RoboDK station: kr30 cnc FIXED BY ALBERT 2.rdk

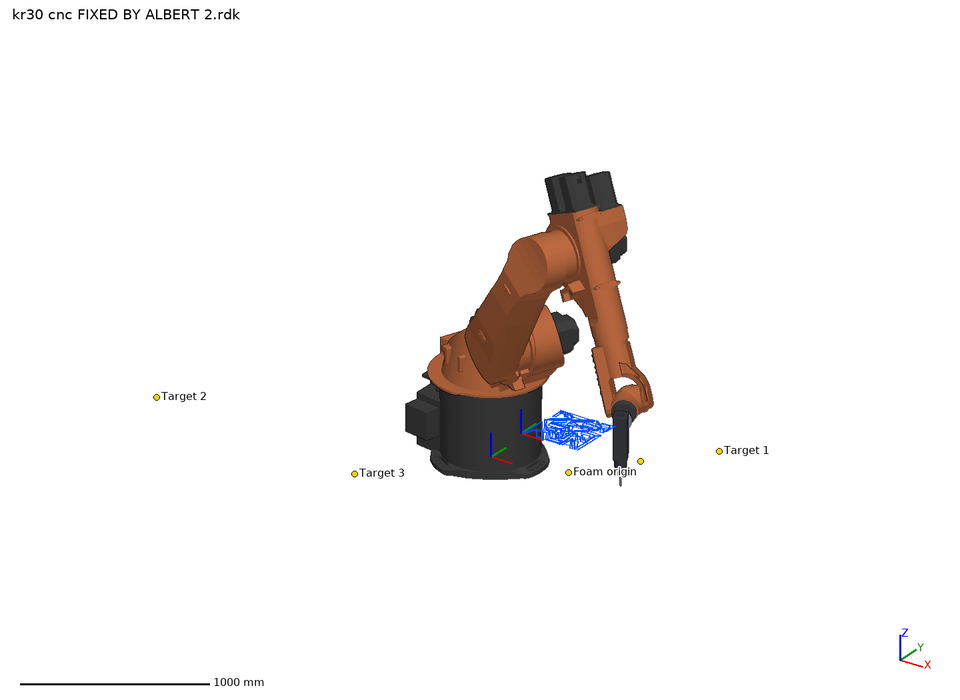
[picture v0: the station drawn from its stored meshes, robots at their saved joint values, targets as dots, program paths as lines]
Station kr30 cnc FIXED BY ALBERT 2. Poses are relative to the parent item; angles as X-Y-Z fixed-axis rotations.
  - frame KUKA KR 30 HA Base at (0, 0, 0) mm
    - robot KUKA KR 30 HA: 6 axes, payload 30 kg, reach 2033 mm, repeatability 0.05 mm, weight 665 kg
        modified DH rows (alpha deg, a mm, theta deg, d mm): 0, 0, 0, 815; -90, 350, 0, 0; 0, 850, -90, 0; -90, 145, 0, 820; 90, 0, 0, 0; -90, 0, 180, 170
        joint limits [-185, -135, -120, -350, -119, -350] to [185, 35, 158, 350, 119, 350]; home [0, -90, 90, 0, 0, 0]; saved at [21.032, -57.583, 122.737, -42.148, -71.052, 16.377]
      - tool 1/2" End Mill TCP, TCP at (337.71, -2.2, 160.57) mm, rotated rx 0 ry 90 rz 0 deg, size 415.8 x 102 x 153.6 mm
    - frame Reference Rhino at (909.29, -1020.53, 801.66) mm
      - object RhinoPart at (150, 150, -300) mm
      - target Target 1 (Cartesian target) at (994.45, 406.4, 10) mm, rotated rx 0 ry 90 rz -60.43 deg; joints [10.582, -19.112, 71.071, -56.398, -66.586, 30.882] of KUKA KR 30 HA
      - target Target 2 (Cartesian target) at (-1810.84, -765.32, 10.08) mm, rotated rx 49.23 ry 89.99 rz -110.09 deg; joints [109.49, -19.11, 71.06, -56.39, -66.58, 30.88] of KUKA KR 30 HA
      - target Target 3 (Cartesian target) at (-425.52, -920.6, 10.08) mm, rotated rx 49.23 ry 89.99 rz -69.31 deg; joints [68.71, -19.11, 71.06, -56.39, -66.58, 30.88] of KUKA KR 30 HA
      - target Foam origin (Cartesian target) at (180.49, 178.32, -252.76) mm, rotated rx -180 ry -0.01 rz -149.04 deg; joints [51.446, -59.335, 121.73, 83.267, -86.48, -27.398] of KUKA KR 30 HA
      - target Foam opposite corner (Cartesian target) at (416.08, 506.55, -249.15) mm, rotated rx -180 ry -0.01 rz -149.04 deg; joints [33.24, -61.647, 125.565, 66.534, -78.959, -23.784] of KUKA KR 30 HA
  - machining project RhinoPart Settings: C:/Users/Julian Ramirez.DESKTOP-JVDE542/Desktop/ELMER SHEET 1 TEST 3.nc | rotZ(0) | rotX(00)*rotY(360) | rotZ(0)
  - object box at (500, 500, 500) mm, size 250 x 250 x 250 mm, geometry from box.sld
  - program RhinoPart (818 instructions, listed below)
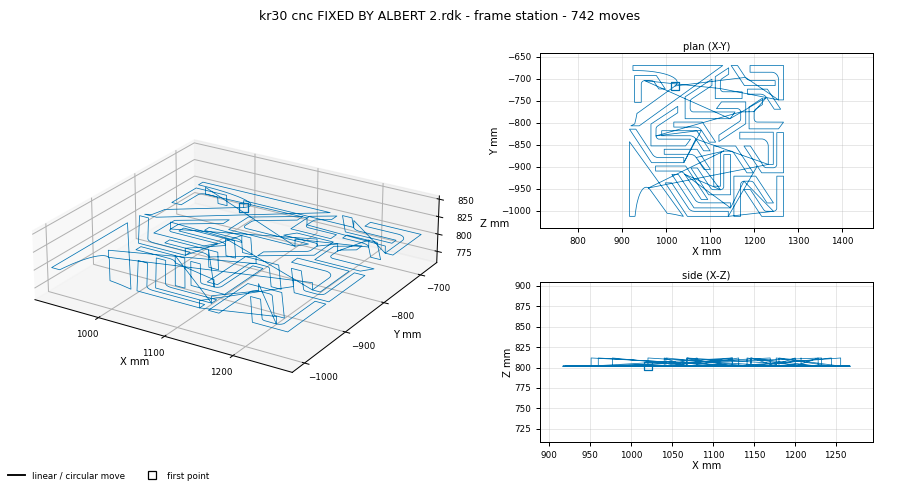
[picture p0: tool path of kr30 cnc FIXED BY ALBERT 2.rdk in frame station, 742 of 742 moves have a stored position in this frame; points joined in program order, loops and branches not executed]

--- program RhinoPart (robot KUKA KR 30 HA) ---
  Smooth(1)
  Set Ref.: Reference Rhino
  Set Tool: 1/2" End Mill TCP
  Show 1/2" End Mill TCP
  Set speed (2000.0 mm/s)
  MoveJ 1 to (111.39, 304.23, 0) mm, rotated rx -180 ry 0 rz 119.57 deg; joints [15.382, -66.233, 141.073, -46.061, -79.352, 10.854]
  MoveL 2 to (111.39, 304.23, 0) mm, rotated rx -180 ry 0 rz 119.57 deg; joints [15.382, -66.233, 141.073, -46.061, -79.352, 10.854]
  MoveL 3 to (111.39, 304.23, 0) mm, rotated rx -180 ry 0 rz 119.57 deg; joints [15.382, -66.233, 141.073, -46.061, -79.352, 10.854]
  Set speed (60.0 mm/s)
  MoveL 4 to (112.73, 305.44, 0) mm, rotated rx 180 ry 0 rz 119.57 deg; joints [15.298, -66.197, 141.001, -46.149, -79.343, 10.896]
  MoveL 5 to (113.84, 306.66, 0) mm, rotated rx -180 ry 0 rz 119.57 deg; joints [15.218, -66.168, 140.944, -46.233, -79.339, 10.931]
  MoveL 6 to (114.75, 307.89, 0) mm, rotated rx 180 ry 0 rz 119.57 deg; joints [15.14, -66.147, 140.903, -46.314, -79.34, 10.96]
  MoveL 7 to (115.44, 309.13, 0) mm, rotated rx 180 ry 0 rz 119.57 deg; joints [15.065, -66.134, 140.877, -46.39, -79.346, 10.983]
  MoveL 8 to (115.92, 310.36, 0) mm, rotated rx -180 ry 0 rz 119.57 deg; joints [14.993, -66.128, 140.867, -46.463, -79.356, 11.001]
  MoveL 9 to (116.19, 311.6, 0) mm, rotated rx -180 ry 0 rz 119.57 deg; joints [14.924, -66.13, 140.871, -46.532, -79.37, 11.012]
  MoveL 10 to (116.26, 312.84, 0) mm, rotated rx -180 ry 0 rz 119.57 deg; joints [14.858, -66.14, 140.89, -46.597, -79.389, 11.017]
  MoveL 11 to (116.12, 314.07, 0) mm, rotated rx -180 ry 0 rz 119.57 deg; joints [14.795, -66.157, 140.923, -46.657, -79.413, 11.017]
  MoveL 12 to (115.78, 315.3, 0) mm, rotated rx -180 ry 0 rz 119.57 deg; joints [14.735, -66.182, 140.972, -46.714, -79.441, 11.01]
  MoveL 13 to (115.23, 316.52, 0) mm, rotated rx -180 ry 0 rz 119.57 deg; joints [14.678, -66.213, 141.034, -46.767, -79.473, 10.998]
  MoveL 14 to (114.49, 317.73, 0) mm, rotated rx -180 ry 0 rz 119.57 deg; joints [14.624, -66.252, 141.111, -46.816, -79.509, 10.98]
  MoveL 15 to (113.55, 318.93, 0) mm, rotated rx 180 ry 0 rz 119.57 deg; joints [14.573, -66.299, 141.202, -46.86, -79.549, 10.956]
  MoveL 16 to (112.41, 320.12, 0) mm, rotated rx -180 ry 0 rz 119.57 deg; joints [14.526, -66.352, 141.307, -46.9, -79.593, 10.926]
  MoveL 17 to (111.07, 321.29, 0) mm, rotated rx 180 ry 0 rz 119.57 deg; joints [14.482, -66.412, 141.425, -46.937, -79.641, 10.891]
  MoveL 18 to (109.54, 322.44, 0) mm, rotated rx 180 ry 0 rz 119.57 deg; joints [14.442, -66.48, 141.557, -46.968, -79.693, 10.85]
  MoveL 19 to (106.83, 324.17, 0) mm, rotated rx 180 ry 0 rz 119.57 deg; joints [14.387, -66.595, 141.785, -47.008, -79.78, 10.776]
  MoveL 20 to (103.93, 325.72, 0) mm, rotated rx 180 ry 0 rz 119.57 deg; joints [14.343, -66.716, 142.023, -47.036, -79.867, 10.697]
  MoveL 21 to (100.95, 327.1, 0) mm, rotated rx 180 ry 0 rz 119.57 deg; joints [14.31, -66.839, 142.264, -47.054, -79.954, 10.615]
  MoveL 22 to (97.98, 328.3, 0) mm, rotated rx 180 ry 0 rz 119.57 deg; joints [14.286, -66.959, 142.5, -47.063, -80.038, 10.533]
  MoveL 23 to (91.45, 330.54, 0) mm, rotated rx -180 ry 0 rz 119.57 deg; joints [14.255, -67.22, 143.011, -47.062, -80.214, 10.352]
  MoveL 24 to (84.62, 332.44, 0) mm, rotated rx 180 ry 0 rz 119.57 deg; joints [14.246, -67.488, 143.537, -47.039, -80.391, 10.162]
  MoveL 25 to (77.71, 334.02, 0) mm, rotated rx 180 ry 0 rz 119.57 deg; joints [14.256, -67.755, 144.061, -46.998, -80.565, 9.97]
  MoveL 26 to (70.95, 335.3, 0) mm, rotated rx -180 ry 0 rz 119.57 deg; joints [14.28, -68.014, 144.569, -46.944, -80.73, 9.781]
  MoveL 27 to (64.72, 336.28, 0) mm, rotated rx -180 ry 0 rz 119.57 deg; joints [14.313, -68.251, 145.032, -46.883, -80.88, 9.608]
  MoveL 28 to (58.43, 337.12, 0) mm, rotated rx -180 ry 0 rz 119.57 deg; joints [14.357, -68.488, 145.496, -46.814, -81.028, 9.434]
  MoveL 29 to (52.12, 337.8, 0) mm, rotated rx -180 ry 0 rz 119.57 deg; joints [14.409, -68.723, 145.958, -46.735, -81.174, 9.259]
  MoveL 30 to (45.84, 338.35, 0) mm, rotated rx -180 ry 0 rz 119.57 deg; joints [14.47, -68.957, 146.414, -46.649, -81.317, 9.086]
  MoveL 31 to (39.9, 338.74, 0) mm, rotated rx 180 ry 0 rz 119.57 deg; joints [14.535, -69.176, 146.843, -46.561, -81.451, 8.922]
  MoveL 32 to (35.07, 338.99, 0) mm, rotated rx 180 ry 0 rz 119.57 deg; joints [14.593, -69.353, 147.189, -46.485, -81.558, 8.79]
  MoveL 33 to (30.23, 339.16, 0) mm, rotated rx 180 ry 0 rz 119.57 deg; joints [14.656, -69.53, 147.535, -46.404, -81.664, 8.657]
  MoveL 34 to (25.39, 339.26, 0) mm, rotated rx -180 ry 0 rz 119.57 deg; joints [14.724, -69.706, 147.878, -46.319, -81.77, 8.525]
  MoveL 35 to (20.56, 339.29, 0) mm, rotated rx 180 ry 0 rz 119.57 deg; joints [14.796, -69.881, 148.22, -46.23, -81.874, 8.393]
  MoveL 36 to (15.58, 339.29, 0) mm, rotated rx 180 ry 0 rz 119.57 deg; joints [14.873, -70.061, 148.57, -46.135, -81.981, 8.258]
  MoveL 37 to (15.58, 350.72, 0) mm, rotated rx -180 ry 0 rz 119.57 deg; joints [14.201, -70.168, 148.779, -46.796, -82.148, 8.276]
  MoveL 38 to (219.85, 350.72, 0) mm, rotated rx 180 ry 0 rz 119.57 deg; joints [11.685, -62.59, 133.888, -50.278, -77.793, 14.278]
  MoveL 39 to (29.95, 213.56, 0) mm, rotated rx 180 ry 0 rz 119.57 deg; joints [21.65, -68.069, 144.677, -39.552, -79.597, 8.481]
  MoveL 40 to (10.8, 213.56, 0) mm, rotated rx -180 ry 0 rz 119.57 deg; joints [22.063, -68.737, 145.985, -39.064, -80.033, 7.996]
  MoveL 41 to (19.53, 217.8, 0) mm, rotated rx -180 ry 0 rz 119.57 deg; joints [21.645, -68.492, 145.505, -39.51, -79.911, 8.22]
  MoveL 42 to (20.98, 223.68, 0) mm, rotated rx -180 ry 0 rz 119.57 deg; joints [21.296, -68.522, 145.564, -39.857, -79.983, 8.262]
  MoveL 43 to (22.33, 229.61, 0) mm, rotated rx 180 ry 0 rz 119.57 deg; joints [20.946, -68.555, 145.629, -40.206, -80.058, 8.303]
  MoveL 44 to (23.58, 235.57, 0) mm, rotated rx -180 ry 0 rz 119.57 deg; joints [20.597, -68.59, 145.698, -40.553, -80.134, 8.341]
  MoveL 45 to (24.71, 241.54, 0) mm, rotated rx 180 ry 0 rz 119.57 deg; joints [20.248, -68.629, 145.773, -40.899, -80.213, 8.376]
  MoveL 46 to (24.55, 241.81, 0) mm, rotated rx 180 ry 0 rz 119.57 deg; joints [20.236, -68.638, 145.791, -40.91, -80.221, 8.372]
  MoveL 47 to (25.65, 242.44, 0) mm, rotated rx -180 ry 0 rz 119.57 deg; joints [20.18, -68.608, 145.732, -40.97, -80.207, 8.402]
  MoveL 48 to (26.73, 243.1, 0) mm, rotated rx 180 ry 0 rz 119.57 deg; joints [20.122, -68.578, 145.674, -41.03, -80.194, 8.43]
  MoveL 49 to (27.79, 243.78, 0) mm, rotated rx 180 ry 0 rz 119.57 deg; joints [20.064, -68.55, 145.618, -41.092, -80.182, 8.458]
  MoveL 50 to (28.82, 244.5, 0) mm, rotated rx 180 ry 0 rz 119.57 deg; joints [20.004, -68.522, 145.565, -41.156, -80.172, 8.486]
  MoveL 51 to (109.85, 303.02, 0) mm, rotated rx 180 ry 0 rz 119.57 deg; joints [15.468, -66.278, 141.161, -45.969, -79.366, 10.807]
  MoveL 52 to (111.39, 304.23, 0) mm, rotated rx -180 ry 0 rz 119.57 deg; joints [15.382, -66.233, 141.073, -46.061, -79.352, 10.854]
  Set speed (2000.0 mm/s)
  MoveL 53 to (111.39, 304.23, 0) mm, rotated rx -180 ry 0 rz 119.57 deg; joints [15.382, -66.233, 141.073, -46.061, -79.352, 10.854]
  MoveL 54 to (111.39, 304.23, 10) mm, rotated rx -180 ry 0 rz 119.57 deg; joints [15.382, -67.039, 141.042, -46.178, -78.772, 11.469]
  Set speed (2000.0 mm/s)
  MoveL 55 to (271.36, 323.77, 0) mm, rotated rx 180 ry 0 rz 119.57 deg; joints [12.449, -60.385, 129.521, -49.903, -76.207, 15.81]
  MoveL 56 to (271.36, 323.77, 0) mm, rotated rx 180 ry 0 rz 119.57 deg; joints [12.449, -60.385, 129.521, -49.903, -76.207, 15.81]
  Set speed (60.0 mm/s)
  MoveL 57 to (253.54, 350.72, 0) mm, rotated rx -180 ry 0 rz 119.57 deg; joints [11.352, -61.296, 131.325, -50.826, -77.072, 15.353]
  MoveL 58 to (238.98, 350.72, 0) mm, rotated rx 180 ry 0 rz 119.57 deg; joints [11.494, -61.857, 132.437, -50.589, -77.384, 14.885]
  MoveL 59 to (269.2, 305, 0) mm, rotated rx 180 ry 0 rz 119.57 deg; joints [13.346, -60.302, 129.357, -49.029, -75.911, 15.659]
  MoveL 60 to (339.09, 305, 0) mm, rotated rx -180 ry 0 rz 119.57 deg; joints [12.617, -57.556, 123.906, -50.298, -74.371, 17.977]
  MoveL 61 to (339.09, 316.43, 0) mm, rotated rx 180 ry 0 rz 119.57 deg; joints [12.112, -57.656, 124.105, -50.776, -74.59, 18.032]
  MoveL 62 to (285.54, 316.43, 0) mm, rotated rx -180 ry 0 rz 119.57 deg; joints [12.643, -59.769, 128.3, -49.827, -75.764, 16.24]
  MoveL 63 to (284.51, 316.46, 0) mm, rotated rx 180 ry 0 rz 119.57 deg; joints [12.652, -59.81, 128.381, -49.81, -75.787, 16.206]
  MoveL 64 to (283.47, 316.55, 0) mm, rotated rx 180 ry 0 rz 119.57 deg; joints [12.659, -59.851, 128.462, -49.796, -75.811, 16.173]
  MoveL 65 to (282.45, 316.7, 0) mm, rotated rx 180 ry 0 rz 119.57 deg; joints [12.663, -59.892, 128.544, -49.784, -75.837, 16.14]
  MoveL 66 to (281.43, 316.91, 0) mm, rotated rx 180 ry 0 rz 119.57 deg; joints [12.664, -59.934, 128.626, -49.775, -75.863, 16.108]
  MoveL 67 to (280.43, 317.18, 0) mm, rotated rx -180 ry 0 rz 119.57 deg; joints [12.662, -59.975, 128.708, -49.769, -75.889, 16.076]
  MoveL 68 to (279.45, 317.5, 0) mm, rotated rx -180 ry 0 rz 119.57 deg; joints [12.657, -60.016, 128.79, -49.766, -75.917, 16.045]
  MoveL 69 to (278.48, 317.88, 0) mm, rotated rx 180 ry 0 rz 119.57 deg; joints [12.649, -60.057, 128.871, -49.766, -75.945, 16.016]
  MoveL 70 to (277.54, 318.32, 0) mm, rotated rx 180 ry 0 rz 119.57 deg; joints [12.638, -60.098, 128.951, -49.769, -75.974, 15.987]
  MoveL 71 to (276.62, 318.82, 0) mm, rotated rx -180 ry 0 rz 119.57 deg; joints [12.625, -60.138, 129.031, -49.775, -76.003, 15.959]
  MoveL 72 to (275.74, 319.38, 0) mm, rotated rx -180 ry 0 rz 119.57 deg; joints [12.608, -60.177, 129.108, -49.784, -76.032, 15.933]
  MoveL 73 to (274.9, 319.98, 0) mm, rotated rx 180 ry 0 rz 119.57 deg; joints [12.589, -60.215, 129.184, -49.797, -76.062, 15.908]
  MoveL 74 to (274.09, 320.64, 0) mm, rotated rx -180 ry 0 rz 119.57 deg; joints [12.566, -60.252, 129.257, -49.812, -76.091, 15.885]
  MoveL 75 to (273.34, 321.35, 0) mm, rotated rx 180 ry 0 rz 119.57 deg; joints [12.541, -60.287, 129.328, -49.83, -76.121, 15.863]
  MoveL 76 to (272.62, 322.11, 0) mm, rotated rx 180 ry 0 rz 119.57 deg; joints [12.513, -60.322, 129.395, -49.852, -76.15, 15.843]
  MoveL 77 to (271.96, 322.92, 0) mm, rotated rx 180 ry 0 rz 119.57 deg; joints [12.483, -60.354, 129.46, -49.876, -76.179, 15.826]
  MoveL 78 to (271.36, 323.77, 0) mm, rotated rx 180 ry 0 rz 119.57 deg; joints [12.449, -60.385, 129.521, -49.903, -76.207, 15.81]
  Set speed (2000.0 mm/s)
  MoveL 79 to (271.36, 323.77, 0) mm, rotated rx 180 ry 0 rz 119.57 deg; joints [12.449, -60.385, 129.521, -49.903, -76.207, 15.81]
  MoveL 80 to (271.36, 323.77, 10) mm, rotated rx -180 ry 0 rz 119.57 deg; joints [12.449, -61.047, 129.494, -50.035, -75.764, 16.354]
  Set speed (2000.0 mm/s)
  MoveL 81 to (346.71, 272.52, 0) mm, rotated rx 180 ry 0 rz 119.57 deg; joints [13.959, -56.946, 122.692, -49.103, -73.566, 18.089]
  MoveL 82 to (346.71, 272.52, 0) mm, rotated rx 180 ry 0 rz 119.57 deg; joints [13.959, -56.946, 122.692, -49.103, -73.566, 18.089]
  Set speed (60.0 mm/s)
  MoveL 83 to (346.71, 318.84, 0) mm, rotated rx -180 ry 0 rz 119.57 deg; joints [11.934, -57.372, 123.54, -51.012, -74.468, 18.305]
  MoveL 84 to (346.64, 320.41, 0) mm, rotated rx -180 ry 0 rz 119.57 deg; joints [11.866, -57.388, 123.571, -51.076, -74.5, 18.31]
  MoveL 85 to (346.44, 321.97, 0) mm, rotated rx 180 ry 0 rz 119.57 deg; joints [11.799, -57.409, 123.614, -51.137, -74.534, 18.31]
  MoveL 86 to (346.1, 323.5, 0) mm, rotated rx 180 ry 0 rz 119.57 deg; joints [11.734, -57.436, 123.666, -51.195, -74.571, 18.306]
  MoveL 87 to (345.63, 324.99, 0) mm, rotated rx 180 ry 0 rz 119.57 deg; joints [11.673, -57.467, 123.728, -51.249, -74.609, 18.297]
  MoveL 88 to (345.02, 326.43, 0) mm, rotated rx 180 ry 0 rz 119.57 deg; joints [11.615, -57.503, 123.8, -51.299, -74.65, 18.284]
  MoveL 89 to (344.29, 327.82, 0) mm, rotated rx -180 ry 0 rz 119.57 deg; joints [11.56, -57.544, 123.881, -51.344, -74.692, 18.265]
  MoveL 90 to (343.43, 329.13, 0) mm, rotated rx -180 ry 0 rz 119.57 deg; joints [11.51, -57.589, 123.971, -51.384, -74.736, 18.242]
  MoveL 91 to (342.44, 330.36, 0) mm, rotated rx -180 ry 0 rz 119.57 deg; joints [11.464, -57.639, 124.069, -51.418, -74.781, 18.215]
  MoveL 92 to (341.34, 331.49, 0) mm, rotated rx 180 ry 0 rz 119.57 deg; joints [11.424, -57.692, 124.175, -51.447, -74.826, 18.182]
  MoveL 93 to (340.15, 332.49, 0) mm, rotated rx -180 ry 0 rz 119.57 deg; joints [11.39, -57.748, 124.286, -51.468, -74.871, 18.146]
  MoveL 94 to (338.86, 333.35, 0) mm, rotated rx -180 ry 0 rz 119.57 deg; joints [11.363, -57.806, 124.402, -51.483, -74.915, 18.107]
  MoveL 95 to (337.5, 334.08, 0) mm, rotated rx -180 ry 0 rz 119.57 deg; joints [11.343, -57.866, 124.522, -51.49, -74.958, 18.064]
  MoveL 96 to (336.07, 334.66, 0) mm, rotated rx 180 ry 0 rz 119.57 deg; joints [11.33, -57.928, 124.644, -51.49, -75, 18.018]
  MoveL 97 to (334.58, 335.09, 0) mm, rotated rx 180 ry 0 rz 119.57 deg; joints [11.324, -57.991, 124.769, -51.483, -75.041, 17.969]
  MoveL 98 to (333.05, 335.35, 0) mm, rotated rx -180 ry 0 rz 119.57 deg; joints [11.326, -58.054, 124.895, -51.468, -75.079, 17.918]
  MoveL 99 to (331.47, 335.44, 0) mm, rotated rx -180 ry 0 rz 119.57 deg; joints [11.336, -58.118, 125.021, -51.445, -75.115, 17.864]
  MoveL 100 to (281.94, 335.44, 0) mm, rotated rx 180 ry 0 rz 119.57 deg; joints [11.799, -60.071, 128.898, -50.605, -76.189, 16.208]
  MoveL 101 to (281.94, 350.72, 0) mm, rotated rx -180 ry 0 rz 119.57 deg; joints [11.086, -60.191, 129.137, -51.287, -76.464, 16.279]
  MoveL 102 to (358.14, 350.72, 0) mm, rotated rx 180 ry 0 rz 119.57 deg; joints [10.429, -57.166, 123.129, -52.535, -74.822, 18.862]
  MoveL 103 to (358.14, 272.52, 0) mm, rotated rx -180 ry 0 rz 119.57 deg; joints [13.837, -56.488, 121.782, -49.326, -73.308, 18.481]
  MoveL 104 to (346.71, 272.52, 0) mm, rotated rx 180 ry 0 rz 119.57 deg; joints [13.959, -56.946, 122.692, -49.103, -73.566, 18.089]
  Set speed (2000.0 mm/s)
  MoveL 105 to (346.71, 272.52, 0) mm, rotated rx 180 ry 0 rz 119.57 deg; joints [13.959, -56.946, 122.692, -49.103, -73.566, 18.089]
  MoveL 106 to (346.71, 272.52, 10) mm, rotated rx -180 ry 0 rz 119.57 deg; joints [13.959, -57.547, 122.667, -49.245, -73.156, 18.585]
  Set speed (2000.0 mm/s)
  MoveL 107 to (214.31, 298.37, 0) mm, rotated rx -180 ry 0 rz 119.57 deg; joints [14.301, -62.342, 133.396, -47.719, -76.996, 13.899]
  MoveL 108 to (214.31, 298.37, 0) mm, rotated rx -180 ry 0 rz 119.57 deg; joints [14.301, -62.342, 133.396, -47.719, -76.996, 13.899]
  Set speed (60.0 mm/s)
  MoveL 109 to (214.27, 299.16, 0) mm, rotated rx -180 ry 0 rz 119.57 deg; joints [14.263, -62.351, 133.414, -47.755, -77.011, 13.901]
  MoveL 110 to (214.27, 313.63, 0) mm, rotated rx 180 ry 0 rz 119.57 deg; joints [13.561, -62.487, 133.683, -48.432, -77.269, 13.955]
  MoveL 111 to (214.33, 314.67, 0) mm, rotated rx -180 ry 0 rz 119.57 deg; joints [13.509, -62.494, 133.697, -48.482, -77.286, 13.961]
  MoveL 112 to (214.51, 315.7, 0) mm, rotated rx 180 ry 0 rz 119.57 deg; joints [13.458, -62.496, 133.702, -48.533, -77.3, 13.97]
  MoveL 113 to (214.81, 316.69, 0) mm, rotated rx -180 ry 0 rz 119.57 deg; joints [13.406, -62.494, 133.697, -48.585, -77.311, 13.983]
  MoveL 114 to (215.22, 317.64, 0) mm, rotated rx -180 ry 0 rz 119.57 deg; joints [13.355, -62.487, 133.684, -48.637, -77.319, 14]
  MoveL 115 to (215.74, 318.53, 0) mm, rotated rx 180 ry 0 rz 119.57 deg; joints [13.305, -62.475, 133.66, -48.688, -77.323, 14.019]
  MoveL 116 to (216.37, 319.35, 0) mm, rotated rx -180 ry 0 rz 119.57 deg; joints [13.258, -62.459, 133.628, -48.738, -77.324, 14.042]
  MoveL 117 to (217.1, 320.09, 0) mm, rotated rx 180 ry 0 rz 119.57 deg; joints [13.214, -62.437, 133.585, -48.785, -77.321, 14.068]
  MoveL 118 to (217.94, 320.73, 0) mm, rotated rx 180 ry 0 rz 119.57 deg; joints [13.173, -62.411, 133.534, -48.83, -77.314, 14.096]
  MoveL 119 to (233.32, 330.89, 0) mm, rotated rx 180 ry 0 rz 119.57 deg; joints [12.51, -61.912, 132.547, -49.572, -77.16, 14.621]
  MoveL 120 to (233.32, 345.45, 0) mm, rotated rx 180 ry 0 rz 119.57 deg; joints [11.806, -62.033, 132.785, -50.251, -77.414, 14.682]
  MoveL 121 to (202.84, 325.31, 0) mm, rotated rx 180 ry 0 rz 119.57 deg; joints [13.121, -63.025, 134.747, -48.782, -77.722, 13.645]
  MoveL 122 to (202.84, 275.58, 0) mm, rotated rx -180 ry 0 rz 119.57 deg; joints [15.551, -62.545, 133.798, -46.439, -76.836, 13.467]
  MoveL 123 to (263.8, 275.58, 0) mm, rotated rx 180 ry 0 rz 119.57 deg; joints [14.771, -60.226, 129.206, -47.626, -75.48, 15.367]
  MoveL 124 to (263.8, 290.86, 0) mm, rotated rx 180 ry 0 rz 119.57 deg; joints [14.064, -60.377, 129.506, -48.302, -75.768, 15.427]
  MoveL 125 to (221.89, 290.86, 0) mm, rotated rx -180 ry 0 rz 119.57 deg; joints [14.569, -61.981, 132.682, -47.514, -76.693, 14.106]
  MoveL 126 to (221.1, 290.91, 0) mm, rotated rx -180 ry 0 rz 119.57 deg; joints [14.576, -62.011, 132.742, -47.501, -76.712, 14.082]
  MoveL 127 to (220.34, 291.04, 0) mm, rotated rx 180 ry 0 rz 119.57 deg; joints [14.58, -62.042, 132.802, -47.492, -76.731, 14.059]
  MoveL 128 to (219.59, 291.25, 0) mm, rotated rx 180 ry 0 rz 119.57 deg; joints [14.579, -62.072, 132.862, -47.488, -76.751, 14.036]
  MoveL 129 to (218.88, 291.54, 0) mm, rotated rx 180 ry 0 rz 119.57 deg; joints [14.574, -62.102, 132.921, -47.488, -76.772, 14.015]
  MoveL 130 to (218.2, 291.9, 0) mm, rotated rx -180 ry 0 rz 119.57 deg; joints [14.565, -62.131, 132.98, -47.492, -76.794, 13.996]
  MoveL 131 to (217.55, 292.34, 0) mm, rotated rx -180 ry 0 rz 119.57 deg; joints [14.552, -62.16, 133.036, -47.5, -76.816, 13.977]
  MoveL 132 to (216.96, 292.84, 0) mm, rotated rx -180 ry 0 rz 119.57 deg; joints [14.535, -62.187, 133.091, -47.512, -76.838, 13.961]
  MoveL 133 to (216.41, 293.4, 0) mm, rotated rx -180 ry 0 rz 119.57 deg; joints [14.515, -62.214, 133.143, -47.527, -76.86, 13.946]
  MoveL 134 to (215.91, 294.02, 0) mm, rotated rx -180 ry 0 rz 119.57 deg; joints [14.491, -62.238, 133.192, -47.547, -76.882, 13.933]
  MoveL 135 to (215.48, 294.67, 0) mm, rotated rx -180 ry 0 rz 119.57 deg; joints [14.465, -62.261, 133.237, -47.569, -76.904, 13.922]
  MoveL 136 to (215.12, 295.36, 0) mm, rotated rx -180 ry 0 rz 119.57 deg; joints [14.436, -62.282, 133.278, -47.594, -76.924, 13.913]
  MoveL 137 to (214.81, 296.09, 0) mm, rotated rx -180 ry 0 rz 119.57 deg; joints [14.405, -62.3, 133.314, -47.622, -76.944, 13.906]
  MoveL 138 to (214.58, 296.83, 0) mm, rotated rx -180 ry 0 rz 119.57 deg; joints [14.372, -62.316, 133.346, -47.653, -76.963, 13.902]
  MoveL 139 to (214.41, 297.6, 0) mm, rotated rx 180 ry 0 rz 119.57 deg; joints [14.337, -62.33, 133.374, -47.685, -76.98, 13.899]
  MoveL 140 to (214.31, 298.37, 0) mm, rotated rx -180 ry 0 rz 119.57 deg; joints [14.301, -62.342, 133.396, -47.719, -76.996, 13.899]
  Set speed (2000.0 mm/s)
  MoveL 141 to (214.31, 298.37, 0) mm, rotated rx -180 ry 0 rz 119.57 deg; joints [14.301, -62.342, 133.396, -47.719, -76.996, 13.899]
  MoveL 142 to (214.31, 298.37, 10) mm, rotated rx -180 ry 0 rz 119.57 deg; joints [14.301, -63.045, 133.368, -47.847, -76.504, 14.456]
  Set speed (2000.0 mm/s)
  MoveL 143 to (41.98, 316.43, 0) mm, rotated rx -180 ry 0 rz 119.57 deg; joints [15.771, -68.882, 146.268, -45.357, -81.064, 8.939]
  MoveL 144 to (41.98, 316.43, 0) mm, rotated rx -180 ry 0 rz 119.57 deg; joints [15.771, -68.882, 146.268, -45.357, -81.064, 8.939]
  Set speed (60.0 mm/s)
  MoveL 145 to (41.2, 316.33, 0) mm, rotated rx -180 ry 0 rz 119.57 deg; joints [15.79, -68.909, 146.321, -45.336, -81.079, 8.917]
  MoveL 146 to (40.44, 316.16, 0) mm, rotated rx -180 ry 0 rz 119.57 deg; joints [15.811, -68.935, 146.372, -45.311, -81.093, 8.896]
  MoveL 147 to (39.69, 315.93, 0) mm, rotated rx 180 ry 0 rz 119.57 deg; joints [15.837, -68.959, 146.42, -45.283, -81.105, 8.875]
  MoveL 148 to (38.97, 315.63, 0) mm, rotated rx 180 ry 0 rz 119.57 deg; joints [15.865, -68.982, 146.464, -45.252, -81.116, 8.855]
  MoveL 149 to (38.28, 315.26, 0) mm, rotated rx 180 ry 0 rz 119.57 deg; joints [15.897, -69.004, 146.506, -45.218, -81.126, 8.836]
  MoveL 150 to (37.62, 314.83, 0) mm, rotated rx -180 ry 0 rz 119.57 deg; joints [15.932, -69.023, 146.544, -45.181, -81.133, 8.817]
  MoveL 151 to (37.01, 314.33, 0) mm, rotated rx 180 ry 0 rz 119.57 deg; joints [15.97, -69.04, 146.577, -45.142, -81.139, 8.799]
  MoveL 152 to (36.44, 313.78, 0) mm, rotated rx -180 ry 0 rz 119.57 deg; joints [16.01, -69.055, 146.605, -45.1, -81.143, 8.783]
  MoveL 153 to (35.94, 313.19, 0) mm, rotated rx 180 ry 0 rz 119.57 deg; joints [16.052, -69.066, 146.629, -45.056, -81.144, 8.769]
  MoveL 154 to (35.51, 312.54, 0) mm, rotated rx 180 ry 0 rz 119.57 deg; joints [16.096, -69.075, 146.646, -45.012, -81.144, 8.756]
  MoveL 155 to (35.14, 311.86, 0) mm, rotated rx 180 ry 0 rz 119.57 deg; joints [16.14, -69.081, 146.658, -44.967, -81.141, 8.745]
  MoveL 156 to (34.85, 311.15, 0) mm, rotated rx 180 ry 0 rz 119.57 deg; joints [16.186, -69.084, 146.664, -44.921, -81.136, 8.736]
  MoveL 157 to (34.64, 310.41, 0) mm, rotated rx -180 ry 0 rz 119.57 deg; joints [16.231, -69.084, 146.664, -44.876, -81.129, 8.729]
  MoveL 158 to (34.51, 309.64, 0) mm, rotated rx -180 ry 0 rz 119.57 deg; joints [16.277, -69.081, 146.657, -44.83, -81.12, 8.724]
  MoveL 159 to (34.47, 308.85, 0) mm, rotated rx 180 ry 0 rz 119.57 deg; joints [16.322, -69.074, 146.644, -44.786, -81.109, 8.722]
  MoveL 160 to (34.47, 266.94, 0) mm, rotated rx -180 ry 0 rz 119.57 deg; joints [18.664, -68.601, 145.719, -42.491, -80.428, 8.661]
  MoveL 161 to (19.18, 266.94, 0) mm, rotated rx 180 ry 0 rz 119.57 deg; joints [18.953, -69.144, 146.781, -42.143, -80.769, 8.26]
  MoveL 162 to (19.18, 327.9, 0) mm, rotated rx 180 ry 0 rz 119.57 deg; joints [15.48, -69.82, 148.1, -45.552, -81.734, 8.338]
  MoveL 163 to (68.91, 327.9, 0) mm, rotated rx 180 ry 0 rz 119.57 deg; joints [14.719, -68.018, 144.578, -46.504, -80.659, 9.707]
  MoveL 164 to (89.06, 297.42, 0) mm, rotated rx 180 ry 0 rz 119.57 deg; joints [16.078, -66.979, 142.539, -45.27, -79.728, 10.204]
  MoveL 165 to (74.5, 297.42, 0) mm, rotated rx -180 ry 0 rz 119.57 deg; joints [16.306, -67.508, 143.577, -44.977, -80.048, 9.798]
  MoveL 166 to (64.33, 312.8, 0) mm, rotated rx -180 ry 0 rz 119.57 deg; joints [15.623, -68.036, 144.613, -45.599, -80.52, 9.547]
  MoveL 167 to (63.69, 313.64, 0) mm, rotated rx -180 ry 0 rz 119.57 deg; joints [15.587, -68.068, 144.675, -45.631, -80.547, 9.531]
  MoveL 168 to (62.96, 314.37, 0) mm, rotated rx 180 ry 0 rz 119.57 deg; joints [15.558, -68.102, 144.741, -45.657, -80.575, 9.512]
  MoveL 169 to (62.14, 315, 0) mm, rotated rx 180 ry 0 rz 119.57 deg; joints [15.536, -68.138, 144.812, -45.675, -80.602, 9.491]
  MoveL 170 to (61.24, 315.52, 0) mm, rotated rx -180 ry 0 rz 119.57 deg; joints [15.521, -68.176, 144.886, -45.686, -80.63, 9.467]
  MoveL 171 to (60.3, 315.93, 0) mm, rotated rx -180 ry 0 rz 119.57 deg; joints [15.512, -68.214, 144.961, -45.689, -80.657, 9.442]
  MoveL 172 to (59.3, 316.23, 0) mm, rotated rx -180 ry 0 rz 119.57 deg; joints [15.511, -68.253, 145.038, -45.686, -80.683, 9.415]
  MoveL 173 to (57.24, 316.47, 0) mm, rotated rx -180 ry 0 rz 119.57 deg; joints [15.53, -68.33, 145.189, -45.659, -80.732, 9.358]
  MoveL 174 to (42.76, 316.47, 0) mm, rotated rx 180 ry 0 rz 119.57 deg; joints [15.757, -68.854, 146.213, -45.374, -81.047, 8.96]
  MoveL 175 to (41.98, 316.43, 0) mm, rotated rx -180 ry 0 rz 119.57 deg; joints [15.771, -68.882, 146.268, -45.357, -81.064, 8.939]
  Set speed (2000.0 mm/s)
  MoveL 176 to (41.98, 316.43, 0) mm, rotated rx -180 ry 0 rz 119.57 deg; joints [15.771, -68.882, 146.268, -45.357, -81.064, 8.939]
  MoveL 177 to (41.98, 316.43, 10) mm, rotated rx 180 ry 0 rz 119.57 deg; joints [15.771, -69.778, 146.234, -45.465, -80.41, 9.61]
  Set speed (2000.0 mm/s)
  MoveL 178 to (236.48, 229.76, 0) mm, rotated rx -180 ry 0 rz 119.57 deg; joints [17.245, -60.767, 130.279, -45.055, -75.213, 14.344]
  MoveL 179 to (236.48, 229.76, 0) mm, rotated rx -180 ry 0 rz 119.57 deg; joints [17.245, -60.767, 130.279, -45.055, -75.213, 14.344]
  Set speed (60.0 mm/s)
  MoveL 180 to (247.91, 245.05, 0) mm, rotated rx -180 ry 0 rz 119.57 deg; joints [16.382, -60.509, 129.767, -45.966, -75.252, 14.751]
  MoveL 181 to (153.31, 245.05, 0) mm, rotated rx 180 ry 0 rz 119.57 deg; joints [17.767, -64.047, 136.766, -43.983, -77.382, 11.905]
  MoveL 182 to (151.76, 245.22, 0) mm, rotated rx -180 ry 0 rz 119.57 deg; joints [17.783, -64.106, 136.883, -43.958, -77.42, 11.861]
  MoveL 183 to (151.01, 245.44, 0) mm, rotated rx 180 ry 0 rz 119.57 deg; joints [17.784, -64.136, 136.942, -43.952, -77.441, 11.84]
  MoveL 184 to (150.3, 245.73, 0) mm, rotated rx -180 ry 0 rz 119.57 deg; joints [17.781, -64.166, 137, -43.951, -77.462, 11.82]
  MoveL 185 to (149.62, 246.09, 0) mm, rotated rx -180 ry 0 rz 119.57 deg; joints [17.774, -64.195, 137.058, -43.953, -77.484, 11.801]
  MoveL 186 to (148.97, 246.52, 0) mm, rotated rx 180 ry 0 rz 119.57 deg; joints [17.762, -64.224, 137.115, -43.96, -77.507, 11.784]
  MoveL 187 to (148.38, 247.03, 0) mm, rotated rx 180 ry 0 rz 119.57 deg; joints [17.747, -64.252, 137.17, -43.972, -77.529, 11.768]
  MoveL 188 to (147.83, 247.59, 0) mm, rotated rx 180 ry 0 rz 119.57 deg; joints [17.728, -64.278, 137.223, -43.987, -77.552, 11.753]
  MoveL 189 to (147.33, 248.2, 0) mm, rotated rx 180 ry 0 rz 119.57 deg; joints [17.705, -64.304, 137.272, -44.006, -77.574, 11.741]
  MoveL 190 to (146.9, 248.86, 0) mm, rotated rx 180 ry 0 rz 119.57 deg; joints [17.679, -64.327, 137.319, -44.028, -77.596, 11.73]
  MoveL 191 to (146.23, 250.27, 0) mm, rotated rx -180 ry 0 rz 119.57 deg; joints [17.619, -64.368, 137.4, -44.082, -77.637, 11.715]
  MoveL 192 to (145.83, 251.78, 0) mm, rotated rx -180 ry 0 rz 119.57 deg; joints [17.55, -64.401, 137.464, -44.147, -77.674, 11.707]
  MoveL 193 to (145.69, 253.35, 0) mm, rotated rx 180 ry 0 rz 119.57 deg; joints [17.475, -64.424, 137.509, -44.219, -77.705, 11.707]
  MoveL 194 to (145.69, 267.82, 0) mm, rotated rx 180 ry 0 rz 119.57 deg; joints [16.749, -64.588, 137.832, -44.922, -77.966, 11.746]
  MoveL 195 to (145.75, 268.86, 0) mm, rotated rx -180 ry 0 rz 119.57 deg; joints [16.695, -64.597, 137.851, -44.974, -77.983, 11.75]
  MoveL 196 to (145.93, 269.89, 0) mm, rotated rx -180 ry 0 rz 119.57 deg; joints [16.641, -64.602, 137.86, -45.028, -77.998, 11.758]
  MoveL 197 to (146.23, 270.88, 0) mm, rotated rx 180 ry 0 rz 119.57 deg; joints [16.587, -64.602, 137.86, -45.082, -78.009, 11.77]
  MoveL 198 to (146.64, 271.83, 0) mm, rotated rx -180 ry 0 rz 119.57 deg; joints [16.533, -64.597, 137.851, -45.137, -78.016, 11.784]
  MoveL 199 to (147.16, 272.72, 0) mm, rotated rx -180 ry 0 rz 119.57 deg; joints [16.48, -64.588, 137.832, -45.191, -78.021, 11.802]
  MoveL 200 to (147.79, 273.54, 0) mm, rotated rx -180 ry 0 rz 119.57 deg; joints [16.429, -64.573, 137.804, -45.244, -78.021, 11.822]
  MoveL 201 to (148.52, 274.28, 0) mm, rotated rx 180 ry 0 rz 119.57 deg; joints [16.381, -64.554, 137.766, -45.295, -78.018, 11.846]
  MoveL 202 to (149.36, 274.91, 0) mm, rotated rx -180 ry 0 rz 119.57 deg; joints [16.337, -64.53, 137.719, -45.343, -78.011, 11.872]
  MoveL 203 to (195.22, 305.23, 0) mm, rotated rx -180 ry 0 rz 119.57 deg; joints [14.203, -63.128, 134.951, -47.688, -77.537, 13.337]
  MoveL 204 to (195.22, 319.79, 0) mm, rotated rx 180 ry 0 rz 119.57 deg; joints [13.484, -63.264, 135.219, -48.383, -77.791, 13.39]
  MoveL 205 to (134.26, 279.5, 0) mm, rotated rx 180 ry 0 rz 119.57 deg; joints [16.329, -65.136, 138.913, -45.264, -78.426, 11.447]
  MoveL 206 to (134.26, 229.76, 0) mm, rotated rx 180 ry 0 rz 119.57 deg; joints [18.837, -64.559, 137.776, -42.833, -77.528, 11.321]
  MoveL 207 to (236.48, 229.76, 0) mm, rotated rx -180 ry 0 rz 119.57 deg; joints [17.245, -60.767, 130.279, -45.055, -75.213, 14.344]
  Set speed (2000.0 mm/s)
  MoveL 208 to (236.48, 229.76, 0) mm, rotated rx -180 ry 0 rz 119.57 deg; joints [17.245, -60.767, 130.279, -45.055, -75.213, 14.344]
  MoveL 209 to (236.48, 229.76, 10) mm, rotated rx -180 ry 0 rz 119.57 deg; joints [17.245, -61.437, 130.252, -45.187, -74.721, 14.855]
  Set speed (2000.0 mm/s)
  MoveL 210 to (319.22, 278.27, 0) mm, rotated rx 180 ry 0 rz 119.57 deg; joints [14.007, -58.094, 124.974, -48.809, -74.295, 17.187]
  MoveL 211 to (319.22, 278.27, 0) mm, rotated rx 180 ry 0 rz 119.57 deg; joints [14.007, -58.094, 124.974, -48.809, -74.295, 17.187]
  Set speed (60.0 mm/s)
  MoveL 212 to (318.61, 279.12, 0) mm, rotated rx 180 ry 0 rz 119.57 deg; joints [13.976, -58.126, 125.038, -48.833, -74.325, 17.17]
  MoveL 213 to (317.95, 279.93, 0) mm, rotated rx -180 ry 0 rz 119.57 deg; joints [13.948, -58.16, 125.105, -48.854, -74.356, 17.151]
  MoveL 214 to (317.24, 280.68, 0) mm, rotated rx -180 ry 0 rz 119.57 deg; joints [13.922, -58.195, 125.176, -48.873, -74.386, 17.131]
  MoveL 215 to (316.48, 281.39, 0) mm, rotated rx -180 ry 0 rz 119.57 deg; joints [13.899, -58.232, 125.249, -48.888, -74.417, 17.109]
  MoveL 216 to (315.68, 282.05, 0) mm, rotated rx 180 ry 0 rz 119.57 deg; joints [13.878, -58.27, 125.324, -48.9, -74.448, 17.085]
  MoveL 217 to (314.83, 282.66, 0) mm, rotated rx -180 ry 0 rz 119.57 deg; joints [13.86, -58.309, 125.402, -48.91, -74.478, 17.059]
  MoveL 218 to (313.95, 283.21, 0) mm, rotated rx 180 ry 0 rz 119.57 deg; joints [13.845, -58.35, 125.482, -48.916, -74.509, 17.032]
  MoveL 219 to (313.04, 283.71, 0) mm, rotated rx 180 ry 0 rz 119.57 deg; joints [13.833, -58.39, 125.563, -48.92, -74.539, 17.004]
  MoveL 220 to (312.09, 284.15, 0) mm, rotated rx -180 ry 0 rz 119.57 deg; joints [13.824, -58.432, 125.645, -48.921, -74.568, 16.975]
  MoveL 221 to (311.13, 284.53, 0) mm, rotated rx -180 ry 0 rz 119.57 deg; joints [13.817, -58.473, 125.728, -48.919, -74.597, 16.944]
  MoveL 222 to (310.15, 284.86, 0) mm, rotated rx 180 ry 0 rz 119.57 deg; joints [13.814, -58.515, 125.811, -48.914, -74.625, 16.913]
  MoveL 223 to (309.14, 285.13, 0) mm, rotated rx -180 ry 0 rz 119.57 deg; joints [13.813, -58.557, 125.894, -48.906, -74.653, 16.881]
  MoveL 224 to (308.13, 285.33, 0) mm, rotated rx 180 ry 0 rz 119.57 deg; joints [13.815, -58.599, 125.977, -48.896, -74.68, 16.848]
  MoveL 225 to (307.1, 285.48, 0) mm, rotated rx 180 ry 0 rz 119.57 deg; joints [13.819, -58.641, 126.06, -48.883, -74.705, 16.815]
  MoveL 226 to (306.07, 285.57, 0) mm, rotated rx -180 ry 0 rz 119.57 deg; joints [13.827, -58.682, 126.142, -48.867, -74.73, 16.781]
  MoveL 227 to (305.03, 285.6, 0) mm, rotated rx 180 ry 0 rz 119.57 deg; joints [13.837, -58.723, 126.224, -48.849, -74.754, 16.747]
  MoveL 228 to (276.12, 285.6, 0) mm, rotated rx -180 ry 0 rz 119.57 deg; joints [14.164, -59.85, 128.461, -48.302, -75.396, 15.802]
  MoveL 229 to (276.12, 297.03, 0) mm, rotated rx 180 ry 0 rz 119.57 deg; joints [13.639, -59.96, 128.678, -48.803, -75.611, 15.849]
  MoveL 230 to (321.38, 297.03, 0) mm, rotated rx -180 ry 0 rz 119.57 deg; joints [13.15, -58.187, 125.16, -49.639, -74.61, 17.341]
  MoveL 231 to (351.59, 251.31, 0) mm, rotated rx -180 ry 0 rz 119.57 deg; joints [14.819, -56.534, 121.872, -48.342, -73.029, 18.164]
  MoveL 232 to (337.03, 251.31, 0) mm, rotated rx 180 ry 0 rz 119.57 deg; joints [14.986, -57.113, 123.025, -48.047, -73.36, 17.67]
  MoveL 233 to (319.22, 278.27, 0) mm, rotated rx 180 ry 0 rz 119.57 deg; joints [14.007, -58.094, 124.974, -48.809, -74.295, 17.187]
  Set speed (2000.0 mm/s)
  MoveL 234 to (319.22, 278.27, 0) mm, rotated rx 180 ry 0 rz 119.57 deg; joints [14.007, -58.094, 124.974, -48.809, -74.295, 17.187]
  MoveL 235 to (319.22, 278.27, 10) mm, rotated rx 180 ry 0 rz 119.57 deg; joints [14.007, -58.714, 124.948, -48.948, -73.87, 17.693]
  Set speed (2000.0 mm/s)
  MoveL 236 to (291.25, 245.76, 0) mm, rotated rx -180 ry 0 rz 119.57 deg; joints [15.784, -58.85, 126.476, -46.886, -74.287, 16.133]
  MoveL 237 to (291.25, 245.76, 0) mm, rotated rx -180 ry 0 rz 119.57 deg; joints [15.784, -58.85, 126.476, -46.886, -74.287, 16.133]
  Set speed (60.0 mm/s)
  MoveL 238 to (291.42, 246.78, 0) mm, rotated rx 180 ry 0 rz 119.57 deg; joints [15.736, -58.854, 126.484, -46.933, -74.303, 16.143]
  MoveL 239 to (291.72, 247.77, 0) mm, rotated rx 180 ry 0 rz 119.57 deg; joints [15.688, -58.854, 126.483, -46.981, -74.316, 16.157]
  MoveL 240 to (292.13, 248.72, 0) mm, rotated rx -180 ry 0 rz 119.57 deg; joints [15.64, -58.848, 126.472, -47.029, -74.325, 16.174]
  MoveL 241 to (292.65, 249.61, 0) mm, rotated rx -180 ry 0 rz 119.57 deg; joints [15.594, -58.838, 126.451, -47.077, -74.331, 16.194]
  MoveL 242 to (293.28, 250.44, 0) mm, rotated rx 180 ry 0 rz 119.57 deg; joints [15.549, -58.822, 126.42, -47.125, -74.333, 16.218]
  MoveL 243 to (294.01, 251.17, 0) mm, rotated rx 180 ry 0 rz 119.57 deg; joints [15.507, -58.801, 126.379, -47.171, -74.331, 16.244]
  MoveL 244 to (294.85, 251.81, 0) mm, rotated rx -180 ry 0 rz 119.57 deg; joints [15.469, -58.776, 126.328, -47.215, -74.325, 16.274]
  MoveL 245 to (310.23, 261.98, 0) mm, rotated rx -180 ry 0 rz 119.57 deg; joints [14.831, -58.282, 125.348, -47.951, -74.178, 16.82]
  MoveL 246 to (310.23, 276.54, 0) mm, rotated rx 180 ry 0 rz 119.57 deg; joints [14.184, -58.43, 125.642, -48.564, -74.463, 16.88]
  MoveL 247 to (279.75, 256.39, 0) mm, rotated rx -180 ry 0 rz 119.57 deg; joints [15.45, -59.41, 127.588, -47.106, -74.755, 15.803]
  MoveL 248 to (279.75, 206.66, 0) mm, rotated rx 180 ry 0 rz 119.57 deg; joints [17.673, -58.84, 126.456, -44.998, -73.763, 15.621]
  MoveL 249 to (346.7, 206.66, 0) mm, rotated rx 180 ry 0 rz 119.57 deg; joints [16.777, -56.225, 121.259, -46.461, -72.218, 17.817]
  MoveL 250 to (358.13, 221.95, 0) mm, rotated rx 180 ry 0 rz 119.57 deg; joints [15.991, -55.949, 120.709, -47.31, -72.274, 18.266]
  MoveL 251 to (298.8, 221.95, 0) mm, rotated rx -180 ry 0 rz 119.57 deg; joints [16.74, -58.287, 125.357, -46.046, -73.637, 16.288]
  MoveL 252 to (298.02, 221.99, 0) mm, rotated rx -180 ry 0 rz 119.57 deg; joints [16.748, -58.318, 125.419, -46.031, -73.656, 16.263]
  MoveL 253 to (297.25, 222.12, 0) mm, rotated rx -180 ry 0 rz 119.57 deg; joints [16.753, -58.349, 125.481, -46.02, -73.676, 16.239]
  MoveL 254 to (296.5, 222.33, 0) mm, rotated rx -180 ry 0 rz 119.57 deg; joints [16.753, -58.381, 125.543, -46.013, -73.697, 16.215]
  MoveL 255 to (295.79, 222.62, 0) mm, rotated rx -180 ry 0 rz 119.57 deg; joints [16.75, -58.412, 125.605, -46.01, -73.72, 16.193]
  MoveL 256 to (295.11, 222.99, 0) mm, rotated rx -180 ry 0 rz 119.57 deg; joints [16.743, -58.442, 125.666, -46.011, -73.743, 16.172]
  MoveL 257 to (294.47, 223.42, 0) mm, rotated rx -180 ry 0 rz 119.57 deg; joints [16.732, -58.472, 125.726, -46.015, -73.766, 16.153]
  MoveL 258 to (293.87, 223.92, 0) mm, rotated rx 180 ry 0 rz 119.57 deg; joints [16.718, -58.501, 125.783, -46.023, -73.79, 16.136]
  MoveL 259 to (293.32, 224.48, 0) mm, rotated rx -180 ry 0 rz 119.57 deg; joints [16.701, -58.529, 125.839, -46.035, -73.814, 16.12]
  MoveL 260 to (292.83, 225.1, 0) mm, rotated rx -180 ry 0 rz 119.57 deg; joints [16.68, -58.555, 125.891, -46.05, -73.838, 16.106]
  MoveL 261 to (292.39, 225.76, 0) mm, rotated rx 180 ry 0 rz 119.57 deg; joints [16.657, -58.58, 125.939, -46.068, -73.861, 16.095]
  MoveL 262 to (292.03, 226.45, 0) mm, rotated rx -180 ry 0 rz 119.57 deg; joints [16.631, -58.602, 125.983, -46.09, -73.883, 16.086]
  MoveL 263 to (291.73, 227.17, 0) mm, rotated rx -180 ry 0 rz 119.57 deg; joints [16.603, -58.622, 126.023, -46.113, -73.904, 16.079]
  MoveL 264 to (291.49, 227.91, 0) mm, rotated rx -180 ry 0 rz 119.57 deg; joints [16.573, -58.64, 126.058, -46.14, -73.925, 16.074]
  MoveL 265 to (291.32, 228.68, 0) mm, rotated rx -180 ry 0 rz 119.57 deg; joints [16.542, -58.655, 126.089, -46.168, -73.944, 16.071]
  MoveL 266 to (291.22, 229.46, 0) mm, rotated rx -180 ry 0 rz 119.57 deg; joints [16.509, -58.668, 126.114, -46.199, -73.962, 16.071]
  MoveL 267 to (291.18, 230.24, 0) mm, rotated rx 180 ry 0 rz 119.57 deg; joints [16.474, -58.678, 126.135, -46.231, -73.979, 16.073]
  MoveL 268 to (291.18, 244.72, 0) mm, rotated rx -180 ry 0 rz 119.57 deg; joints [15.831, -58.841, 126.458, -46.84, -74.267, 16.127]
  MoveL 269 to (291.25, 245.76, 0) mm, rotated rx -180 ry 0 rz 119.57 deg; joints [15.784, -58.85, 126.476, -46.886, -74.287, 16.133]
  Set speed (2000.0 mm/s)
  MoveL 270 to (291.25, 245.76, 0) mm, rotated rx -180 ry 0 rz 119.57 deg; joints [15.784, -58.85, 126.476, -46.886, -74.287, 16.133]
  MoveL 271 to (291.25, 245.76, 10) mm, rotated rx -180 ry 0 rz 119.57 deg; joints [15.784, -59.483, 126.449, -47.023, -73.836, 16.635]
  Set speed (2000.0 mm/s)
  MoveL 272 to (260.67, 245.16, 0) mm, rotated rx 180 ry 0 rz 119.57 deg; joints [16.206, -60.022, 128.802, -46.233, -74.966, 15.153]
  MoveL 273 to (260.67, 245.16, 0) mm, rotated rx 180 ry 0 rz 119.57 deg; joints [16.206, -60.022, 128.802, -46.233, -74.966, 15.153]
  Set speed (60.0 mm/s)
  MoveL 274 to (260.57, 245.93, 0) mm, rotated rx -180 ry 0 rz 119.57 deg; joints [16.172, -60.035, 128.827, -46.265, -74.984, 15.152]
  MoveL 275 to (260.4, 246.7, 0) mm, rotated rx 180 ry 0 rz 119.57 deg; joints [16.139, -60.05, 128.857, -46.295, -75.002, 15.15]
  MoveL 276 to (260.16, 247.45, 0) mm, rotated rx 180 ry 0 rz 119.57 deg; joints [16.108, -60.067, 128.891, -46.322, -75.022, 15.145]
  MoveL 277 to (259.86, 248.17, 0) mm, rotated rx 180 ry 0 rz 119.57 deg; joints [16.079, -60.087, 128.93, -46.348, -75.043, 15.138]
  MoveL 278 to (259.49, 248.86, 0) mm, rotated rx 180 ry 0 rz 119.57 deg; joints [16.053, -60.109, 128.973, -46.37, -75.065, 15.129]
  MoveL 279 to (259.06, 249.52, 0) mm, rotated rx -180 ry 0 rz 119.57 deg; joints [16.028, -60.132, 129.02, -46.39, -75.087, 15.118]
  MoveL 280 to (258.57, 250.13, 0) mm, rotated rx -180 ry 0 rz 119.57 deg; joints [16.006, -60.158, 129.071, -46.407, -75.11, 15.104]
  MoveL 281 to (258.02, 250.69, 0) mm, rotated rx -180 ry 0 rz 119.57 deg; joints [15.988, -60.185, 129.125, -46.42, -75.133, 15.089]
  MoveL 282 to (257.42, 251.19, 0) mm, rotated rx -180 ry 0 rz 119.57 deg; joints [15.973, -60.214, 129.181, -46.43, -75.157, 15.072]
  MoveL 283 to (256.78, 251.63, 0) mm, rotated rx -180 ry 0 rz 119.57 deg; joints [15.961, -60.243, 129.239, -46.436, -75.179, 15.053]
  MoveL 284 to (256.1, 251.99, 0) mm, rotated rx 180 ry 0 rz 119.57 deg; joints [15.954, -60.273, 129.299, -46.438, -75.202, 15.033]
  MoveL 285 to (255.38, 252.28, 0) mm, rotated rx 180 ry 0 rz 119.57 deg; joints [15.95, -60.303, 129.359, -46.436, -75.223, 15.012]
  MoveL 286 to (254.64, 252.49, 0) mm, rotated rx 180 ry 0 rz 119.57 deg; joints [15.95, -60.334, 129.42, -46.431, -75.244, 14.989]
  MoveL 287 to (253.87, 252.62, 0) mm, rotated rx 180 ry 0 rz 119.57 deg; joints [15.954, -60.365, 129.481, -46.421, -75.264, 14.965]
  MoveL 288 to (253.08, 252.67, 0) mm, rotated rx 180 ry 0 rz 119.57 deg; joints [15.962, -60.396, 129.542, -46.407, -75.283, 14.941]
  MoveL 289 to (205.51, 252.67, 0) mm, rotated rx 180 ry 0 rz 119.57 deg; joints [16.613, -62.197, 133.109, -45.435, -76.352, 13.473]
  MoveL 290 to (216.94, 267.96, 0) mm, rotated rx -180 ry 0 rz 119.57 deg; joints [15.727, -61.933, 132.588, -46.366, -76.382, 13.872]
  MoveL 291 to (272.13, 267.96, 0) mm, rotated rx 180 ry 0 rz 119.57 deg; joints [15.019, -59.827, 128.414, -47.455, -75.149, 15.603]
  MoveL 292 to (272.13, 218.22, 0) mm, rotated rx -180 ry 0 rz 119.57 deg; joints [17.266, -59.272, 127.314, -45.319, -74.172, 15.419]
  MoveL 293 to (211.17, 177.93, 0) mm, rotated rx 180 ry 0 rz 119.57 deg; joints [20.012, -61.061, 130.861, -42.219, -74.758, 13.417]
  MoveL 294 to (211.17, 192.49, 0) mm, rotated rx -180 ry 0 rz 119.57 deg; joints [19.346, -61.255, 131.245, -42.856, -75.053, 13.459]
  MoveL 295 to (257.04, 222.8, 0) mm, rotated rx -180 ry 0 rz 119.57 deg; joints [17.271, -59.904, 128.568, -45.19, -74.608, 14.959]
  MoveL 296 to (257.87, 223.44, 0) mm, rotated rx -180 ry 0 rz 119.57 deg; joints [17.23, -59.88, 128.52, -45.236, -74.602, 14.988]
  MoveL 297 to (258.61, 224.18, 0) mm, rotated rx -180 ry 0 rz 119.57 deg; joints [17.187, -59.861, 128.481, -45.283, -74.6, 15.013]
  MoveL 298 to (259.24, 225, 0) mm, rotated rx -180 ry 0 rz 119.57 deg; joints [17.141, -59.846, 128.453, -45.332, -74.602, 15.036]
  MoveL 299 to (259.76, 225.89, 0) mm, rotated rx -180 ry 0 rz 119.57 deg; joints [17.093, -59.837, 128.434, -45.381, -74.608, 15.055]
  MoveL 300 to (260.17, 226.84, 0) mm, rotated rx -180 ry 0 rz 119.57 deg; joints [17.045, -59.832, 128.425, -45.431, -74.617, 15.071]
  MoveL 301 to (260.46, 227.83, 0) mm, rotated rx -180 ry 0 rz 119.57 deg; joints [16.996, -59.833, 128.426, -45.48, -74.63, 15.084]
  MoveL 302 to (260.7, 229.9, 0) mm, rotated rx -180 ry 0 rz 119.57 deg; joints [16.899, -59.848, 128.455, -45.574, -74.666, 15.099]
  MoveL 303 to (260.7, 244.37, 0) mm, rotated rx -180 ry 0 rz 119.57 deg; joints [16.241, -60.012, 128.782, -46.2, -74.95, 15.151]
  MoveL 304 to (260.67, 245.16, 0) mm, rotated rx 180 ry 0 rz 119.57 deg; joints [16.206, -60.022, 128.802, -46.233, -74.966, 15.153]
  Set speed (2000.0 mm/s)
  MoveL 305 to (260.67, 245.16, 0) mm, rotated rx 180 ry 0 rz 119.57 deg; joints [16.206, -60.022, 128.802, -46.233, -74.966, 15.153]
  MoveL 306 to (260.67, 245.16, 10) mm, rotated rx 180 ry 0 rz 119.57 deg; joints [16.206, -60.677, 128.775, -46.368, -74.495, 15.664]
  Set speed (2000.0 mm/s)
  MoveL 307 to (67.97, 190.64, 0) mm, rotated rx -180 ry 0 rz 119.57 deg; joints [22.05, -66.412, 141.424, -39.347, -78.303, 9.437]
  MoveL 308 to (67.97, 190.64, 0) mm, rotated rx -180 ry 0 rz 119.57 deg; joints [22.05, -66.412, 141.424, -39.347, -78.303, 9.437]
  Set speed (60.0 mm/s)
  MoveL 309 to (67.93, 191.43, 0) mm, rotated rx 180 ry 0 rz 119.57 deg; joints [22.011, -66.424, 141.448, -39.385, -78.319, 9.437]
  MoveL 310 to (67.93, 205.9, 0) mm, rotated rx -180 ry 0 rz 119.57 deg; joints [21.269, -66.627, 141.847, -40.106, -78.591, 9.459]
  MoveL 311 to (68.17, 207.97, 0) mm, rotated rx 180 ry 0 rz 119.57 deg; joints [21.158, -66.646, 141.886, -40.216, -78.624, 9.469]
  MoveL 312 to (68.47, 208.96, 0) mm, rotated rx 180 ry 0 rz 119.57 deg; joints [21.101, -66.65, 141.892, -40.273, -78.636, 9.478]
  MoveL 313 to (68.88, 209.91, 0) mm, rotated rx -180 ry 0 rz 119.57 deg; joints [21.044, -66.648, 141.889, -40.33, -78.644, 9.49]
  MoveL 314 to (69.4, 210.8, 0) mm, rotated rx -180 ry 0 rz 119.57 deg; joints [20.987, -66.642, 141.876, -40.388, -78.649, 9.505]
  MoveL 315 to (70.03, 211.62, 0) mm, rotated rx -180 ry 0 rz 119.57 deg; joints [20.933, -66.631, 141.854, -40.444, -78.649, 9.523]
  MoveL 316 to (70.76, 212.36, 0) mm, rotated rx -180 ry 0 rz 119.57 deg; joints [20.88, -66.615, 141.823, -40.499, -78.646, 9.544]
  MoveL 317 to (71.6, 213, 0) mm, rotated rx 180 ry 0 rz 119.57 deg; joints [20.831, -66.593, 141.781, -40.552, -78.639, 9.567]
  MoveL 318 to (117.46, 243.31, 0) mm, rotated rx -180 ry 0 rz 119.57 deg; joints [18.441, -65.335, 139.306, -43.119, -78.156, 10.879]
  MoveL 319 to (117.46, 257.87, 0) mm, rotated rx -180 ry 0 rz 119.57 deg; joints [17.698, -65.508, 139.646, -43.84, -78.418, 10.913]
  MoveL 320 to (56.5, 217.58, 0) mm, rotated rx -180 ry 0 rz 119.57 deg; joints [20.892, -67.19, 142.953, -40.417, -79.067, 9.175]
  MoveL 321 to (56.5, 167.84, 0) mm, rotated rx -180 ry 0 rz 119.57 deg; joints [23.451, -66.478, 141.555, -37.926, -78.128, 9.108]
  MoveL 322 to (135.21, 167.84, 0) mm, rotated rx -180 ry 0 rz 119.57 deg; joints [21.839, -63.695, 136.07, -39.939, -76.31, 11.208]
  MoveL 323 to (146.64, 183.13, 0) mm, rotated rx -180 ry 0 rz 119.57 deg; joints [20.894, -63.498, 135.682, -40.923, -76.351, 11.562]
  MoveL 324 to (75.55, 183.13, 0) mm, rotated rx -180 ry 0 rz 119.57 deg; joints [22.274, -66.037, 140.686, -39.169, -77.985, 9.625]
  MoveL 325 to (74.77, 183.17, 0) mm, rotated rx -180 ry 0 rz 119.57 deg; joints [22.288, -66.065, 140.742, -39.151, -78.004, 9.604]
  MoveL 326 to (74, 183.3, 0) mm, rotated rx -180 ry 0 rz 119.57 deg; joints [22.298, -66.094, 140.799, -39.138, -78.024, 9.584]
  MoveL 327 to (73.25, 183.52, 0) mm, rotated rx -180 ry 0 rz 119.57 deg; joints [22.302, -66.123, 140.857, -39.13, -78.046, 9.565]
  MoveL 328 to (72.54, 183.81, 0) mm, rotated rx -180 ry 0 rz 119.57 deg; joints [22.303, -66.152, 140.914, -39.126, -78.068, 9.547]
  MoveL 329 to (71.86, 184.17, 0) mm, rotated rx 180 ry 0 rz 119.57 deg; joints [22.298, -66.182, 140.972, -39.126, -78.09, 9.529]
  MoveL 330 to (71.22, 184.61, 0) mm, rotated rx -180 ry 0 rz 119.57 deg; joints [22.29, -66.211, 141.029, -39.131, -78.113, 9.513]
  MoveL 331 to (70.62, 185.11, 0) mm, rotated rx -180 ry 0 rz 119.57 deg; joints [22.277, -66.239, 141.084, -39.141, -78.137, 9.498]
  MoveL 332 to (70.07, 185.67, 0) mm, rotated rx -180 ry 0 rz 119.57 deg; joints [22.26, -66.266, 141.138, -39.155, -78.16, 9.485]
  MoveL 333 to (69.57, 186.28, 0) mm, rotated rx 180 ry 0 rz 119.57 deg; joints [22.239, -66.293, 141.19, -39.172, -78.183, 9.473]
  MoveL 334 to (69.14, 186.94, 0) mm, rotated rx -180 ry 0 rz 119.57 deg; joints [22.214, -66.317, 141.238, -39.194, -78.206, 9.462]
  MoveL 335 to (68.78, 187.63, 0) mm, rotated rx -180 ry 0 rz 119.57 deg; joints [22.187, -66.34, 141.283, -39.219, -78.227, 9.454]
  MoveL 336 to (68.48, 188.35, 0) mm, rotated rx 180 ry 0 rz 119.57 deg; joints [22.156, -66.361, 141.324, -39.247, -78.248, 9.447]
  MoveL 337 to (68.24, 189.1, 0) mm, rotated rx 180 ry 0 rz 119.57 deg; joints [22.123, -66.38, 141.362, -39.277, -78.268, 9.442]
  MoveL 338 to (68.07, 189.86, 0) mm, rotated rx -180 ry 0 rz 119.57 deg; joints [22.088, -66.397, 141.395, -39.311, -78.286, 9.439]
  MoveL 339 to (67.97, 190.64, 0) mm, rotated rx -180 ry 0 rz 119.57 deg; joints [22.05, -66.412, 141.424, -39.347, -78.303, 9.437]
  Set speed (2000.0 mm/s)
  MoveL 340 to (67.97, 190.64, 0) mm, rotated rx -180 ry 0 rz 119.57 deg; joints [22.05, -66.412, 141.424, -39.347, -78.303, 9.437]
  MoveL 341 to (67.97, 190.64, 10) mm, rotated rx -180 ry 0 rz 119.57 deg; joints [22.05, -67.223, 141.392, -39.461, -77.652, 9.984]
  Set speed (2000.0 mm/s)
  MoveL 342 to (171.32, 203.38, 0) mm, rotated rx -180 ry 0 rz 119.57 deg; joints [19.493, -62.87, 134.44, -42.433, -76.183, 12.316]
  MoveL 343 to (171.32, 203.38, 0) mm, rotated rx -180 ry 0 rz 119.57 deg; joints [19.493, -62.87, 134.44, -42.433, -76.183, 12.316]
  Set speed (60.0 mm/s)
  MoveL 344 to (170.71, 204.23, 0) mm, rotated rx -180 ry 0 rz 119.57 deg; joints [19.463, -62.903, 134.506, -42.458, -76.213, 12.301]
  MoveL 345 to (170.05, 205.04, 0) mm, rotated rx -180 ry 0 rz 119.57 deg; joints [19.436, -62.938, 134.575, -42.48, -76.244, 12.284]
  MoveL 346 to (169.34, 205.79, 0) mm, rotated rx 180 ry 0 rz 119.57 deg; joints [19.412, -62.974, 134.646, -42.498, -76.275, 12.265]
  MoveL 347 to (168.58, 206.5, 0) mm, rotated rx 180 ry 0 rz 119.57 deg; joints [19.391, -63.011, 134.719, -42.514, -76.306, 12.245]
  MoveL 348 to (167.78, 207.16, 0) mm, rotated rx -180 ry 0 rz 119.57 deg; joints [19.373, -63.049, 134.794, -42.526, -76.337, 12.224]
  MoveL 349 to (166.94, 207.77, 0) mm, rotated rx -180 ry 0 rz 119.57 deg; joints [19.358, -63.087, 134.87, -42.534, -76.368, 12.201]
  MoveL 350 to (166.05, 208.32, 0) mm, rotated rx -180 ry 0 rz 119.57 deg; joints [19.346, -63.127, 134.948, -42.54, -76.399, 12.177]
  MoveL 351 to (165.14, 208.82, 0) mm, rotated rx -180 ry 0 rz 119.57 deg; joints [19.337, -63.167, 135.027, -42.542, -76.43, 12.152]
  MoveL 352 to (164.2, 209.26, 0) mm, rotated rx 180 ry 0 rz 119.57 deg; joints [19.332, -63.207, 135.107, -42.541, -76.46, 12.126]
  MoveL 353 to (163.23, 209.65, 0) mm, rotated rx 180 ry 0 rz 119.57 deg; joints [19.33, -63.247, 135.186, -42.537, -76.489, 12.099]
  MoveL 354 to (162.25, 209.97, 0) mm, rotated rx -180 ry 0 rz 119.57 deg; joints [19.331, -63.287, 135.266, -42.529, -76.518, 12.071]
  MoveL 355 to (161.25, 210.24, 0) mm, rotated rx 180 ry 0 rz 119.57 deg; joints [19.335, -63.328, 135.345, -42.519, -76.546, 12.043]
  MoveL 356 to (160.23, 210.44, 0) mm, rotated rx 180 ry 0 rz 119.57 deg; joints [19.342, -63.367, 135.424, -42.506, -76.573, 12.014]
  MoveL 357 to (159.21, 210.59, 0) mm, rotated rx 180 ry 0 rz 119.57 deg; joints [19.353, -63.407, 135.502, -42.489, -76.599, 11.985]
  MoveL 358 to (158.17, 210.68, 0) mm, rotated rx -180 ry 0 rz 119.57 deg; joints [19.366, -63.446, 135.579, -42.47, -76.624, 11.956]
  MoveL 359 to (157.13, 210.71, 0) mm, rotated rx -180 ry 0 rz 119.57 deg; joints [19.382, -63.484, 135.654, -42.447, -76.649, 11.926]
  MoveL 360 to (108.51, 210.71, 0) mm, rotated rx 180 ry 0 rz 119.57 deg; joints [20.244, -65.245, 139.129, -41.321, -77.756, 10.561]
  MoveL 361 to (108.51, 222.14, 0) mm, rotated rx 180 ry 0 rz 119.57 deg; joints [19.669, -65.395, 139.423, -41.878, -77.97, 10.584]
  MoveL 362 to (173.48, 222.14, 0) mm, rotated rx -180 ry 0 rz 119.57 deg; joints [18.56, -63.028, 134.754, -43.345, -76.496, 12.429]
  MoveL 363 to (203.7, 176.42, 0) mm, rotated rx -180 ry 0 rz 119.57 deg; joints [20.206, -61.318, 131.37, -41.978, -74.9, 13.191]
  MoveL 364 to (189.14, 176.42, 0) mm, rotated rx -180 ry 0 rz 119.57 deg; joints [20.455, -61.855, 132.433, -41.634, -75.237, 12.763]
  MoveL 365 to (171.32, 203.38, 0) mm, rotated rx -180 ry 0 rz 119.57 deg; joints [19.493, -62.87, 134.44, -42.433, -76.183, 12.316]
  Set speed (2000.0 mm/s)
  MoveL 366 to (171.32, 203.38, 0) mm, rotated rx -180 ry 0 rz 119.57 deg; joints [19.493, -62.87, 134.44, -42.433, -76.183, 12.316]
  MoveL 367 to (171.32, 203.38, 10) mm, rotated rx -180 ry 0 rz 119.57 deg; joints [19.493, -63.585, 134.411, -42.559, -75.634, 12.835]
  Set speed (2000.0 mm/s)
  MoveL 368 to (131.27, 129.74, 0) mm, rotated rx 180 ry 0 rz 119.57 deg; joints [23.716, -63.264, 135.219, -38.107, -75.622, 11.021]
  MoveL 369 to (131.27, 129.74, 0) mm, rotated rx 180 ry 0 rz 119.57 deg; joints [23.716, -63.264, 135.219, -38.107, -75.622, 11.021]
  Set speed (60.0 mm/s)
  MoveL 370 to (131.27, 141.17, 0) mm, rotated rx 180 ry 0 rz 119.57 deg; joints [23.181, -63.44, 135.567, -38.622, -75.859, 11.044]
  MoveL 371 to (74.34, 141.17, 0) mm, rotated rx -180 ry 0 rz 119.57 deg; joints [24.383, -65.445, 139.522, -37.118, -77.184, 9.529]
  MoveL 372 to (70.22, 141.65, 0) mm, rotated rx 180 ry 0 rz 119.57 deg; joints [24.451, -65.596, 139.819, -37.029, -77.289, 9.424]
  MoveL 373 to (68.24, 142.24, 0) mm, rotated rx 180 ry 0 rz 119.57 deg; joints [24.467, -65.674, 139.973, -37.003, -77.347, 9.374]
  MoveL 374 to (66.33, 143.06, 0) mm, rotated rx -180 ry 0 rz 119.57 deg; joints [24.469, -65.753, 140.129, -36.991, -77.408, 9.326]
  MoveL 375 to (64.53, 144.12, 0) mm, rotated rx -180 ry 0 rz 119.57 deg; joints [24.457, -65.832, 140.285, -36.992, -77.471, 9.281]
  MoveL 376 to (62.88, 145.38, 0) mm, rotated rx -180 ry 0 rz 119.57 deg; joints [24.432, -65.91, 140.436, -37.008, -77.535, 9.241]
  MoveL 377 to (61.41, 146.85, 0) mm, rotated rx -180 ry 0 rz 119.57 deg; joints [24.392, -65.984, 140.582, -37.038, -77.599, 9.205]
  MoveL 378 to (60.15, 148.51, 0) mm, rotated rx 180 ry 0 rz 119.57 deg; joints [24.339, -66.054, 140.72, -37.084, -77.661, 9.175]
  MoveL 379 to (22.19, 205.94, 0) mm, rotated rx 180 ry 0 rz 119.57 deg; joints [22.223, -68.233, 144.998, -38.957, -79.636, 8.276]
  MoveL 380 to (7.63, 205.94, 0) mm, rotated rx -180 ry 0 rz 119.57 deg; joints [22.545, -68.739, 145.988, -38.579, -79.968, 7.911]
  MoveL 381 to (57.99, 129.74, 0) mm, rotated rx 180 ry 0 rz 119.57 deg; joints [25.313, -65.828, 140.276, -36.127, -77.331, 9.095]
  MoveL 382 to (131.27, 129.74, 0) mm, rotated rx 180 ry 0 rz 119.57 deg; joints [23.716, -63.264, 135.219, -38.107, -75.622, 11.021]
  Set speed (2000.0 mm/s)
  MoveL 383 to (131.27, 129.74, 0) mm, rotated rx 180 ry 0 rz 119.57 deg; joints [23.716, -63.264, 135.219, -38.107, -75.622, 11.021]
  MoveL 384 to (131.27, 129.74, 10) mm, rotated rx -180 ry 0 rz 119.57 deg; joints [23.716, -63.989, 135.19, -38.229, -75.029, 11.502]
  Set speed (2000.0 mm/s)
  MoveL 385 to (158.56, 183.68, 0) mm, rotated rx -180 ry 0 rz 119.57 deg; joints [20.652, -63.073, 134.842, -41.234, -76.088, 11.9]
  MoveL 386 to (158.56, 183.68, 0) mm, rotated rx -180 ry 0 rz 119.57 deg; joints [20.652, -63.073, 134.842, -41.234, -76.088, 11.9]
  Set speed (60.0 mm/s)
  MoveL 387 to (157.95, 184.53, 0) mm, rotated rx -180 ry 0 rz 119.57 deg; joints [20.622, -63.107, 134.909, -41.258, -76.119, 11.885]
  MoveL 388 to (157.29, 185.34, 0) mm, rotated rx 180 ry 0 rz 119.57 deg; joints [20.596, -63.142, 134.978, -41.279, -76.15, 11.868]
  MoveL 389 to (156.58, 186.09, 0) mm, rotated rx 180 ry 0 rz 119.57 deg; joints [20.573, -63.178, 135.049, -41.297, -76.181, 11.85]
  MoveL 390 to (155.82, 186.8, 0) mm, rotated rx 180 ry 0 rz 119.57 deg; joints [20.552, -63.215, 135.123, -41.311, -76.212, 11.83]
  MoveL 391 to (155.02, 187.46, 0) mm, rotated rx -180 ry 0 rz 119.57 deg; joints [20.535, -63.253, 135.198, -41.323, -76.244, 11.809]
  MoveL 392 to (154.18, 188.07, 0) mm, rotated rx 180 ry 0 rz 119.57 deg; joints [20.521, -63.292, 135.275, -41.33, -76.275, 11.786]
  MoveL 393 to (153.3, 188.62, 0) mm, rotated rx -180 ry 0 rz 119.57 deg; joints [20.511, -63.332, 135.353, -41.335, -76.306, 11.763]
  MoveL 394 to (152.37, 189.13, 0) mm, rotated rx -180 ry 0 rz 119.57 deg; joints [20.503, -63.372, 135.433, -41.336, -76.337, 11.738]
  MoveL 395 to (151.44, 189.56, 0) mm, rotated rx 180 ry 0 rz 119.57 deg; joints [20.499, -63.412, 135.512, -41.334, -76.367, 11.712]
  MoveL 396 to (150.48, 189.95, 0) mm, rotated rx -180 ry 0 rz 119.57 deg; joints [20.498, -63.452, 135.591, -41.329, -76.397, 11.686]
  MoveL 397 to (149.49, 190.27, 0) mm, rotated rx -180 ry 0 rz 119.57 deg; joints [20.5, -63.492, 135.671, -41.321, -76.426, 11.659]
  MoveL 398 to (148.49, 190.54, 0) mm, rotated rx 180 ry 0 rz 119.57 deg; joints [20.505, -63.532, 135.75, -41.309, -76.454, 11.631]
  MoveL 399 to (147.47, 190.75, 0) mm, rotated rx 180 ry 0 rz 119.57 deg; joints [20.513, -63.572, 135.828, -41.295, -76.482, 11.603]
  MoveL 400 to (146.44, 190.9, 0) mm, rotated rx -180 ry 0 rz 119.57 deg; joints [20.525, -63.611, 135.906, -41.277, -76.508, 11.574]
  MoveL 401 to (145.41, 190.99, 0) mm, rotated rx -180 ry 0 rz 119.57 deg; joints [20.539, -63.65, 135.982, -41.257, -76.534, 11.545]
  MoveL 402 to (144.37, 191.02, 0) mm, rotated rx -180 ry 0 rz 119.57 deg; joints [20.556, -63.688, 136.057, -41.234, -76.558, 11.516]
  MoveL 403 to (80.97, 191.02, 0) mm, rotated rx -180 ry 0 rz 119.57 deg; joints [21.766, -65.958, 140.531, -39.692, -78.012, 9.781]
  MoveL 404 to (80.97, 202.45, 0) mm, rotated rx -180 ry 0 rz 119.57 deg; joints [21.187, -66.117, 140.845, -40.254, -78.229, 9.8]
  MoveL 405 to (160.71, 202.45, 0) mm, rotated rx 180 ry 0 rz 119.57 deg; joints [19.719, -63.246, 135.184, -42.146, -76.407, 12.008]
  MoveL 406 to (190.93, 156.73, 0) mm, rotated rx 180 ry 0 rz 119.57 deg; joints [21.329, -61.513, 131.756, -40.811, -74.792, 12.763]
  MoveL 407 to (176.37, 156.73, 0) mm, rotated rx -180 ry 0 rz 119.57 deg; joints [21.591, -62.045, 132.81, -40.454, -75.13, 12.343]
  MoveL 408 to (158.56, 183.68, 0) mm, rotated rx -180 ry 0 rz 119.57 deg; joints [20.652, -63.073, 134.842, -41.234, -76.088, 11.9]
  Set speed (2000.0 mm/s)
  MoveL 409 to (158.56, 183.68, 0) mm, rotated rx -180 ry 0 rz 119.57 deg; joints [20.652, -63.073, 134.842, -41.234, -76.088, 11.9]
  MoveL 410 to (158.56, 183.68, 10) mm, rotated rx -180 ry 0 rz 119.57 deg; joints [20.652, -63.794, 134.813, -41.359, -75.525, 12.41]
  Set speed (2000.0 mm/s)
  MoveL 411 to (323.38, 125.76, 0) mm, rotated rx 180 ry 0 rz 119.57 deg; joints [20.479, -56.07, 120.95, -42.772, -71.008, 16.755]
  MoveL 412 to (323.38, 125.76, 0) mm, rotated rx 180 ry 0 rz 119.57 deg; joints [20.479, -56.07, 120.95, -42.772, -71.008, 16.755]
  Set speed (60.0 mm/s)
  MoveL 413 to (334.81, 125.76, 0) mm, rotated rx -180 ry 0 rz 119.57 deg; joints [20.305, -55.624, 120.062, -43.052, -70.735, 17.131]
  MoveL 414 to (334.81, 199.04, 0) mm, rotated rx 180 ry 0 rz 119.57 deg; joints [17.253, -56.604, 122.012, -45.898, -72.333, 17.388]
  MoveL 415 to (258.61, 199.04, 0) mm, rotated rx -180 ry 0 rz 119.57 deg; joints [18.316, -59.554, 127.873, -44.209, -74.094, 14.928]
  MoveL 416 to (258.61, 183.75, 0) mm, rotated rx -180 ry 0 rz 119.57 deg; joints [18.996, -59.358, 127.484, -43.564, -73.78, 14.878]
  MoveL 417 to (308.14, 183.75, 0) mm, rotated rx 180 ry 0 rz 119.57 deg; joints [18.269, -57.456, 123.706, -44.69, -72.63, 16.453]
  MoveL 418 to (309.71, 183.66, 0) mm, rotated rx -180 ry 0 rz 119.57 deg; joints [18.25, -57.394, 123.582, -44.722, -72.591, 16.504]
  MoveL 419 to (311.25, 183.4, 0) mm, rotated rx -180 ry 0 rz 119.57 deg; joints [18.24, -57.33, 123.457, -44.747, -72.55, 16.554]
  MoveL 420 to (312.74, 182.98, 0) mm, rotated rx 180 ry 0 rz 119.57 deg; joints [18.237, -57.267, 123.331, -44.763, -72.507, 16.601]
  MoveL 421 to (314.17, 182.4, 0) mm, rotated rx -180 ry 0 rz 119.57 deg; joints [18.241, -57.204, 123.205, -44.772, -72.461, 16.645]
  MoveL 422 to (315.53, 181.67, 0) mm, rotated rx -180 ry 0 rz 119.57 deg; joints [18.253, -57.142, 123.081, -44.774, -72.414, 16.687]
  MoveL 423 to (316.81, 180.8, 0) mm, rotated rx 180 ry 0 rz 119.57 deg; joints [18.272, -57.08, 122.96, -44.769, -72.365, 16.726]
  MoveL 424 to (318.01, 179.8, 0) mm, rotated rx -180 ry 0 rz 119.57 deg; joints [18.298, -57.021, 122.841, -44.756, -72.316, 16.762]
  MoveL 425 to (319.11, 178.68, 0) mm, rotated rx 180 ry 0 rz 119.57 deg; joints [18.33, -56.963, 122.727, -44.736, -72.266, 16.794]
  MoveL 426 to (320.09, 177.45, 0) mm, rotated rx -180 ry 0 rz 119.57 deg; joints [18.369, -56.909, 122.618, -44.71, -72.217, 16.822]
  MoveL 427 to (320.95, 176.13, 0) mm, rotated rx 180 ry 0 rz 119.57 deg; joints [18.412, -56.858, 122.518, -44.678, -72.169, 16.846]
  MoveL 428 to (321.69, 174.75, 0) mm, rotated rx -180 ry 0 rz 119.57 deg; joints [18.46, -56.811, 122.425, -44.64, -72.122, 16.865]
  MoveL 429 to (322.29, 173.31, 0) mm, rotated rx 180 ry 0 rz 119.57 deg; joints [18.513, -56.769, 122.34, -44.597, -72.077, 16.88]
  MoveL 430 to (322.76, 171.81, 0) mm, rotated rx 180 ry 0 rz 119.57 deg; joints [18.569, -56.731, 122.265, -44.548, -72.034, 16.89]
  MoveL 431 to (323.1, 170.28, 0) mm, rotated rx 180 ry 0 rz 119.57 deg; joints [18.629, -56.698, 122.198, -44.496, -71.993, 16.896]
  MoveL 432 to (323.31, 168.73, 0) mm, rotated rx -180 ry 0 rz 119.57 deg; joints [18.691, -56.669, 122.142, -44.439, -71.955, 16.897]
  MoveL 433 to (323.38, 167.16, 0) mm, rotated rx -180 ry 0 rz 119.57 deg; joints [18.756, -56.646, 122.095, -44.379, -71.919, 16.894]
  MoveL 434 to (323.38, 125.76, 0) mm, rotated rx 180 ry 0 rz 119.57 deg; joints [20.479, -56.07, 120.95, -42.772, -71.008, 16.755]
  Set speed (2000.0 mm/s)
  MoveL 435 to (323.38, 125.76, 0) mm, rotated rx 180 ry 0 rz 119.57 deg; joints [20.479, -56.07, 120.95, -42.772, -71.008, 16.755]
  MoveL 436 to (323.38, 125.76, 10) mm, rotated rx -180 ry 0 rz 119.57 deg; joints [20.479, -56.658, 120.925, -42.917, -70.558, 17.197]
  Set speed (2000.0 mm/s)
  MoveL 437 to (50.74, 72.13, 0) mm, rotated rx -180 ry 0 rz 119.57 deg; joints [28.25, -65.083, 138.809, -33.244, -76.279, 8.837]
  MoveL 438 to (50.74, 72.13, 0) mm, rotated rx -180 ry 0 rz 119.57 deg; joints [28.25, -65.083, 138.809, -33.244, -76.279, 8.837]
  Set speed (60.0 mm/s)
  MoveL 439 to (49.73, 72.75, 0) mm, rotated rx 180 ry 0 rz 119.57 deg; joints [28.246, -65.128, 138.898, -33.242, -76.317, 8.813]
  MoveL 440 to (48.69, 73.25, 0) mm, rotated rx -180 ry 0 rz 119.57 deg; joints [28.249, -65.172, 138.985, -33.233, -76.352, 8.788]
  MoveL 441 to (47.63, 73.6, 0) mm, rotated rx -180 ry 0 rz 119.57 deg; joints [28.259, -65.215, 139.068, -33.218, -76.385, 8.763]
  MoveL 442 to (46.55, 73.81, 0) mm, rotated rx 180 ry 0 rz 119.57 deg; joints [28.277, -65.255, 139.147, -33.194, -76.415, 8.737]
  MoveL 443 to (45.44, 73.85, 0) mm, rotated rx 180 ry 0 rz 119.57 deg; joints [28.303, -65.293, 139.223, -33.163, -76.442, 8.71]
  MoveL 444 to (44.31, 73.72, 0) mm, rotated rx -180 ry 0 rz 119.57 deg; joints [28.337, -65.329, 139.293, -33.123, -76.466, 8.682]
  MoveL 445 to (43.16, 73.42, 0) mm, rotated rx -180 ry 0 rz 119.57 deg; joints [28.381, -65.362, 139.358, -33.075, -76.486, 8.653]
  MoveL 446 to (41.99, 72.92, 0) mm, rotated rx -180 ry 0 rz 119.57 deg; joints [28.434, -65.392, 139.418, -33.017, -76.502, 8.624]
  MoveL 447 to (40.81, 72.22, 0) mm, rotated rx 180 ry 0 rz 119.57 deg; joints [28.498, -65.419, 139.471, -32.949, -76.515, 8.595]
  MoveL 448 to (39.61, 71.3, 0) mm, rotated rx -180 ry 0 rz 119.57 deg; joints [28.571, -65.443, 139.517, -32.871, -76.523, 8.564]
  MoveL 449 to (38.39, 70.17, 0) mm, rotated rx 180 ry 0 rz 119.57 deg; joints [28.656, -65.463, 139.557, -32.782, -76.527, 8.534]
  MoveL 450 to (36.66, 68.16, 0) mm, rotated rx -180 ry 0 rz 119.57 deg; joints [28.795, -65.484, 139.598, -32.638, -76.523, 8.489]
  MoveL 451 to (35.1, 65.94, 0) mm, rotated rx -180 ry 0 rz 119.57 deg; joints [28.94, -65.495, 139.62, -32.489, -76.511, 8.449]
  MoveL 452 to (33.71, 63.6, 0) mm, rotated rx 180 ry 0 rz 119.57 deg; joints [29.086, -65.498, 139.626, -32.34, -76.492, 8.412]
  MoveL 453 to (32.5, 61.26, 0) mm, rotated rx 180 ry 0 rz 119.57 deg; joints [29.228, -65.495, 139.62, -32.196, -76.469, 8.38]
  MoveL 454 to (31.29, 58.64, 0) mm, rotated rx 180 ry 0 rz 119.57 deg; joints [29.383, -65.486, 139.603, -32.04, -76.439, 8.348]
  MoveL 455 to (30.17, 55.91, 0) mm, rotated rx 180 ry 0 rz 119.57 deg; joints [29.54, -65.472, 139.575, -31.882, -76.405, 8.318]
  MoveL 456 to (28.18, 50.23, 0) mm, rotated rx -180 ry 0 rz 119.57 deg; joints [29.858, -65.431, 139.494, -31.563, -76.325, 8.263]
  MoveL 457 to (26.49, 44.44, 0) mm, rotated rx 180 ry 0 rz 119.57 deg; joints [30.172, -65.376, 139.386, -31.25, -76.235, 8.216]
  MoveL 458 to (25.09, 38.8, 0) mm, rotated rx 180 ry 0 rz 119.57 deg; joints [30.47, -65.313, 139.263, -30.954, -76.14, 8.176]
  MoveL 459 to (24.66, 36.87, 0) mm, rotated rx -180 ry 0 rz 119.57 deg; joints [30.571, -65.29, 139.217, -30.854, -76.107, 8.163]
  MoveL 460 to (23.26, 29.74, 0) mm, rotated rx 180 ry 0 rz 119.57 deg; joints [30.936, -65.197, 139.033, -30.493, -75.977, 8.121]
  MoveL 461 to (22.08, 22.46, 0) mm, rotated rx -180 ry 0 rz 119.57 deg; joints [31.301, -65.091, 138.825, -30.134, -75.837, 8.084]
  MoveL 462 to (21.12, 15.1, 0) mm, rotated rx 180 ry 0 rz 119.57 deg; joints [31.661, -64.975, 138.596, -29.78, -75.689, 8.051]
  MoveL 463 to (20.36, 7.75, 0) mm, rotated rx -180 ry 0 rz 119.57 deg; joints [32.013, -64.851, 138.352, -29.436, -75.535, 8.023]
  MoveL 464 to (19.05, 7.63, 0) mm, rotated rx -180 ry 0 rz 119.57 deg; joints [32.055, -64.891, 138.431, -29.387, -75.563, 7.992]
  MoveL 465 to (7.62, 7.63, 0) mm, rotated rx -180 ry 0 rz 119.57 deg; joints [32.379, -65.262, 139.161, -29.011, -75.833, 7.73]
  MoveL 466 to (7.62, 177.44, 0) mm, rotated rx -180 ry 0 rz 119.57 deg; joints [24.066, -68.315, 145.159, -37.093, -79.439, 7.89]
  MoveL 467 to (130.27, 7.63, 0) mm, rotated rx -180 ry 0 rz 119.57 deg; joints [29.182, -61.167, 131.072, -32.865, -72.917, 10.746]
  MoveL 468 to (121.21, 9.76, 0) mm, rotated rx -180 ry 0 rz 119.57 deg; joints [29.308, -61.52, 131.77, -32.679, -73.185, 10.513]
  MoveL 469 to (111.98, 11.68, 0) mm, rotated rx 180 ry 0 rz 119.57 deg; joints [29.448, -61.873, 132.469, -32.479, -73.451, 10.277]
  MoveL 470 to (102.71, 13.32, 0) mm, rotated rx 180 ry 0 rz 119.57 deg; joints [29.604, -62.221, 133.157, -32.265, -73.711, 10.041]
  MoveL 471 to (93.49, 14.59, 0) mm, rotated rx -180 ry 0 rz 119.57 deg; joints [29.777, -62.559, 133.825, -32.037, -73.961, 9.809]
  MoveL 472 to (55.32, 67.43, 0) mm, rotated rx -180 ry 0 rz 119.57 deg; joints [28.354, -64.843, 138.336, -33.17, -76.068, 8.943]
  MoveL 473 to (53.59, 69.59, 0) mm, rotated rx -180 ry 0 rz 119.57 deg; joints [28.297, -64.941, 138.528, -33.215, -76.157, 8.904]
  MoveL 474 to (51.72, 71.39, 0) mm, rotated rx -180 ry 0 rz 119.57 deg; joints [28.26, -65.036, 138.717, -33.24, -76.24, 8.86]
  MoveL 475 to (50.74, 72.13, 0) mm, rotated rx -180 ry 0 rz 119.57 deg; joints [28.25, -65.083, 138.809, -33.244, -76.279, 8.837]
  Set speed (2000.0 mm/s)
  MoveL 476 to (50.74, 72.13, 0) mm, rotated rx -180 ry 0 rz 119.57 deg; joints [28.25, -65.083, 138.809, -33.244, -76.279, 8.837]
  MoveL 477 to (50.74, 72.13, 10) mm, rotated rx -180 ry 0 rz 119.57 deg; joints [28.25, -65.855, 138.778, -33.355, -75.608, 9.291]
  Set speed (2000.0 mm/s)
  MoveL 478 to (222.19, 156.18, 0) mm, rotated rx -180 ry 0 rz 119.57 deg; joints [20.81, -60.351, 129.454, -41.545, -74.052, 13.684]
  MoveL 479 to (222.19, 156.18, 0) mm, rotated rx -180 ry 0 rz 119.57 deg; joints [20.81, -60.351, 129.454, -41.545, -74.052, 13.684]
  Set speed (60.0 mm/s)
  MoveL 480 to (222.97, 156.21, 0) mm, rotated rx 180 ry 0 rz 119.57 deg; joints [20.795, -60.322, 129.397, -41.565, -74.035, 13.707]
  MoveL 481 to (237.45, 156.21, 0) mm, rotated rx 180 ry 0 rz 119.57 deg; joints [20.552, -59.782, 128.326, -41.913, -73.697, 14.143]
  MoveL 482 to (239.51, 155.97, 0) mm, rotated rx -180 ry 0 rz 119.57 deg; joints [20.528, -59.702, 128.166, -41.952, -73.644, 14.205]
  MoveL 483 to (240.5, 155.67, 0) mm, rotated rx -180 ry 0 rz 119.57 deg; joints [20.525, -59.66, 128.084, -41.963, -73.614, 14.235]
  MoveL 484 to (241.45, 155.26, 0) mm, rotated rx -180 ry 0 rz 119.57 deg; joints [20.527, -59.619, 128.002, -41.969, -73.583, 14.262]
  MoveL 485 to (242.35, 154.74, 0) mm, rotated rx -180 ry 0 rz 119.57 deg; joints [20.536, -59.578, 127.921, -41.968, -73.551, 14.288]
  MoveL 486 to (243.17, 154.11, 0) mm, rotated rx -180 ry 0 rz 119.57 deg; joints [20.55, -59.539, 127.842, -41.962, -73.519, 14.311]
  MoveL 487 to (243.9, 153.38, 0) mm, rotated rx -180 ry 0 rz 119.57 deg; joints [20.57, -59.501, 127.767, -41.949, -73.486, 14.331]
  MoveL 488 to (244.54, 152.54, 0) mm, rotated rx -180 ry 0 rz 119.57 deg; joints [20.596, -59.465, 127.696, -41.929, -73.453, 14.348]
  MoveL 489 to (274.85, 106.68, 0) mm, rotated rx 180 ry 0 rz 119.57 deg; joints [22.057, -57.647, 124.087, -40.82, -71.737, 15.147]
  MoveL 490 to (289.41, 106.68, 0) mm, rotated rx 180 ry 0 rz 119.57 deg; joints [21.812, -57.094, 122.987, -41.188, -71.389, 15.603]
  MoveL 491 to (249.12, 167.64, 0) mm, rotated rx -180 ry 0 rz 119.57 deg; joints [19.857, -59.502, 127.769, -42.669, -73.665, 14.534]
  MoveL 492 to (199.39, 167.64, 0) mm, rotated rx -180 ry 0 rz 119.57 deg; joints [20.682, -61.356, 131.445, -41.492, -74.82, 13.04]
  MoveL 493 to (199.39, 76.2, 0) mm, rotated rx -180 ry 0 rz 119.57 deg; joints [24.741, -59.955, 128.668, -37.626, -72.851, 12.805]
  MoveL 494 to (214.68, 76.2, 0) mm, rotated rx 180 ry 0 rz 119.57 deg; joints [24.441, -59.399, 127.565, -38.037, -72.486, 13.248]
  MoveL 495 to (214.68, 148.59, 0) mm, rotated rx 180 ry 0 rz 119.57 deg; joints [21.278, -60.522, 129.792, -41.04, -74.068, 13.439]
  MoveL 496 to (214.72, 149.38, 0) mm, rotated rx 180 ry 0 rz 119.57 deg; joints [21.242, -60.531, 129.811, -41.074, -74.084, 13.442]
  MoveL 497 to (214.85, 150.15, 0) mm, rotated rx -180 ry 0 rz 119.57 deg; joints [21.205, -60.538, 129.823, -41.11, -74.097, 13.448]
  MoveL 498 to (215.06, 150.89, 0) mm, rotated rx -180 ry 0 rz 119.57 deg; joints [21.168, -60.54, 129.829, -41.147, -74.108, 13.456]
  MoveL 499 to (215.35, 151.6, 0) mm, rotated rx -180 ry 0 rz 119.57 deg; joints [21.131, -60.54, 129.828, -41.185, -74.116, 13.467]
  MoveL 500 to (215.72, 152.29, 0) mm, rotated rx -180 ry 0 rz 119.57 deg; joints [21.094, -60.536, 129.82, -41.222, -74.122, 13.48]
  MoveL 501 to (216.15, 152.93, 0) mm, rotated rx 180 ry 0 rz 119.57 deg; joints [21.058, -60.529, 129.807, -41.26, -74.125, 13.494]
  MoveL 502 to (216.65, 153.53, 0) mm, rotated rx 180 ry 0 rz 119.57 deg; joints [21.023, -60.519, 129.787, -41.298, -74.126, 13.511]
  MoveL 503 to (217.21, 154.08, 0) mm, rotated rx -180 ry 0 rz 119.57 deg; joints [20.988, -60.506, 129.761, -41.335, -74.124, 13.529]
  MoveL 504 to (217.83, 154.57, 0) mm, rotated rx 180 ry 0 rz 119.57 deg; joints [20.956, -60.49, 129.73, -41.371, -74.12, 13.549]
  MoveL 505 to (218.49, 155, 0) mm, rotated rx -180 ry 0 rz 119.57 deg; joints [20.925, -60.472, 129.694, -41.405, -74.114, 13.57]
  MoveL 506 to (219.18, 155.37, 0) mm, rotated rx -180 ry 0 rz 119.57 deg; joints [20.897, -60.452, 129.653, -41.438, -74.105, 13.591]
  MoveL 507 to (219.9, 155.67, 0) mm, rotated rx -180 ry 0 rz 119.57 deg; joints [20.871, -60.429, 129.608, -41.468, -74.095, 13.614]
  MoveL 508 to (220.65, 155.9, 0) mm, rotated rx -180 ry 0 rz 119.57 deg; joints [20.848, -60.405, 129.56, -41.496, -74.083, 13.637]
  MoveL 509 to (221.41, 156.07, 0) mm, rotated rx 180 ry 0 rz 119.57 deg; joints [20.827, -60.379, 129.508, -41.522, -74.068, 13.66]
  MoveL 510 to (222.19, 156.18, 0) mm, rotated rx -180 ry 0 rz 119.57 deg; joints [20.81, -60.351, 129.454, -41.545, -74.052, 13.684]
  Set speed (2000.0 mm/s)
  MoveL 511 to (222.19, 156.18, 0) mm, rotated rx -180 ry 0 rz 119.57 deg; joints [20.81, -60.351, 129.454, -41.545, -74.052, 13.684]
  MoveL 512 to (222.19, 156.18, 10) mm, rotated rx -180 ry 0 rz 119.57 deg; joints [20.81, -61.013, 129.427, -41.678, -73.537, 14.16]
  Set speed (2000.0 mm/s)
  MoveL 513 to (159.39, 141.46, 0) mm, rotated rx -180 ry 0 rz 119.57 deg; joints [22.614, -62.436, 133.583, -39.355, -75.21, 11.824]
  MoveL 514 to (159.39, 141.46, 0) mm, rotated rx -180 ry 0 rz 119.57 deg; joints [22.614, -62.436, 133.583, -39.355, -75.21, 11.824]
  Set speed (60.0 mm/s)
  MoveL 515 to (158.78, 142.31, 0) mm, rotated rx -180 ry 0 rz 119.57 deg; joints [22.586, -62.471, 133.652, -39.377, -75.242, 11.809]
  MoveL 516 to (158.12, 143.12, 0) mm, rotated rx -180 ry 0 rz 119.57 deg; joints [22.561, -62.507, 133.723, -39.396, -75.274, 11.792]
  MoveL 517 to (157.41, 143.88, 0) mm, rotated rx -180 ry 0 rz 119.57 deg; joints [22.54, -62.544, 133.796, -39.412, -75.306, 11.774]
  MoveL 518 to (156.65, 144.58, 0) mm, rotated rx -180 ry 0 rz 119.57 deg; joints [22.522, -62.582, 133.871, -39.424, -75.338, 11.755]
  MoveL 519 to (155.85, 145.24, 0) mm, rotated rx 180 ry 0 rz 119.57 deg; joints [22.507, -62.621, 133.948, -39.433, -75.371, 11.734]
  MoveL 520 to (155, 145.85, 0) mm, rotated rx 180 ry 0 rz 119.57 deg; joints [22.495, -62.66, 134.026, -39.439, -75.403, 11.711]
  MoveL 521 to (154.12, 146.4, 0) mm, rotated rx -180 ry 0 rz 119.57 deg; joints [22.486, -62.7, 134.105, -39.441, -75.435, 11.688]
  MoveL 522 to (153.2, 146.9, 0) mm, rotated rx 180 ry 0 rz 119.57 deg; joints [22.48, -62.741, 134.185, -39.44, -75.467, 11.663]
  MoveL 523 to (152.26, 147.34, 0) mm, rotated rx -180 ry 0 rz 119.57 deg; joints [22.478, -62.781, 134.265, -39.436, -75.498, 11.638]
  MoveL 524 to (151.3, 147.73, 0) mm, rotated rx -180 ry 0 rz 119.57 deg; joints [22.479, -62.821, 134.345, -39.429, -75.528, 11.612]
  MoveL 525 to (150.31, 148.05, 0) mm, rotated rx 180 ry 0 rz 119.57 deg; joints [22.483, -62.862, 134.424, -39.419, -75.558, 11.585]
  MoveL 526 to (149.31, 148.32, 0) mm, rotated rx -180 ry 0 rz 119.57 deg; joints [22.49, -62.902, 134.504, -39.405, -75.586, 11.558]
  MoveL 527 to (148.3, 148.53, 0) mm, rotated rx 180 ry 0 rz 119.57 deg; joints [22.499, -62.941, 134.582, -39.389, -75.614, 11.53]
  MoveL 528 to (147.27, 148.67, 0) mm, rotated rx 180 ry 0 rz 119.57 deg; joints [22.512, -62.98, 134.659, -39.37, -75.641, 11.502]
  MoveL 529 to (146.24, 148.76, 0) mm, rotated rx -180 ry 0 rz 119.57 deg; joints [22.528, -63.019, 134.735, -39.347, -75.667, 11.473]
  MoveL 530 to (145.2, 148.79, 0) mm, rotated rx 180 ry 0 rz 119.57 deg; joints [22.547, -63.057, 134.81, -39.323, -75.692, 11.444]
  MoveL 531 to (86.73, 148.79, 0) mm, rotated rx -180 ry 0 rz 119.57 deg; joints [23.741, -65.131, 138.904, -37.809, -77.05, 9.864]
  MoveL 532 to (86.73, 160.22, 0) mm, rotated rx -180 ry 0 rz 119.57 deg; joints [23.182, -65.305, 139.247, -38.351, -77.279, 9.883]
  MoveL 533 to (161.54, 160.22, 0) mm, rotated rx -180 ry 0 rz 119.57 deg; joints [21.702, -62.635, 133.975, -40.245, -75.546, 11.929]
  MoveL 534 to (191.76, 114.5, 0) mm, rotated rx -180 ry 0 rz 119.57 deg; joints [23.215, -60.851, 130.444, -39.017, -73.878, 12.68]
  MoveL 535 to (177.2, 114.5, 0) mm, rotated rx -180 ry 0 rz 119.57 deg; joints [23.495, -61.379, 131.49, -38.639, -74.221, 12.264]
  MoveL 536 to (159.39, 141.46, 0) mm, rotated rx -180 ry 0 rz 119.57 deg; joints [22.614, -62.436, 133.583, -39.355, -75.21, 11.824]
  Set speed (2000.0 mm/s)
  MoveL 537 to (159.39, 141.46, 0) mm, rotated rx -180 ry 0 rz 119.57 deg; joints [22.614, -62.436, 133.583, -39.355, -75.21, 11.824]
  MoveL 538 to (159.39, 141.46, 10) mm, rotated rx 180 ry 0 rz 119.57 deg; joints [22.614, -63.142, 133.555, -39.48, -74.643, 12.307]
  Set speed (2000.0 mm/s)
  MoveL 539 to (214.78, 68.13, 0) mm, rotated rx 180 ry 0 rz 119.57 deg; joints [24.783, -59.26, 127.289, -37.715, -72.3, 13.23]
  MoveL 540 to (214.78, 68.13, 0) mm, rotated rx 180 ry 0 rz 119.57 deg; joints [24.783, -59.26, 127.289, -37.715, -72.3, 13.23]
  Set speed (60.0 mm/s)
  MoveL 541 to (214, 68.1, 0) mm, rotated rx -180 ry 0 rz 119.57 deg; joints [24.8, -59.288, 127.345, -37.692, -72.318, 13.207]
  MoveL 542 to (199.52, 68.1, 0) mm, rotated rx -180 ry 0 rz 119.57 deg; joints [25.087, -59.814, 128.388, -37.299, -72.664, 12.789]
  MoveL 543 to (197.46, 68.34, 0) mm, rotated rx -180 ry 0 rz 119.57 deg; joints [25.118, -59.892, 128.544, -37.253, -72.719, 12.73]
  MoveL 544 to (196.47, 68.63, 0) mm, rotated rx -180 ry 0 rz 119.57 deg; joints [25.125, -59.933, 128.625, -37.238, -72.749, 12.703]
  MoveL 545 to (195.52, 69.04, 0) mm, rotated rx 180 ry 0 rz 119.57 deg; joints [25.127, -59.975, 128.707, -37.229, -72.781, 12.676]
  MoveL 546 to (194.63, 69.56, 0) mm, rotated rx -180 ry 0 rz 119.57 deg; joints [25.122, -60.016, 128.789, -37.226, -72.814, 12.652]
  MoveL 547 to (193.81, 70.19, 0) mm, rotated rx 180 ry 0 rz 119.57 deg; joints [25.112, -60.056, 128.869, -37.229, -72.848, 12.63]
  MoveL 548 to (193.07, 70.93, 0) mm, rotated rx -180 ry 0 rz 119.57 deg; joints [25.095, -60.095, 128.946, -37.239, -72.882, 12.611]
  MoveL 549 to (192.43, 71.76, 0) mm, rotated rx -180 ry 0 rz 119.57 deg; joints [25.072, -60.132, 129.02, -37.256, -72.916, 12.595]
  MoveL 550 to (162.12, 117.63, 0) mm, rotated rx -180 ry 0 rz 119.57 deg; joints [23.651, -61.972, 132.664, -38.38, -74.643, 11.846]
  MoveL 551 to (147.56, 117.63, 0) mm, rotated rx -180 ry 0 rz 119.57 deg; joints [23.943, -62.493, 133.695, -37.998, -74.985, 11.442]
  MoveL 552 to (187.85, 56.67, 0) mm, rotated rx -180 ry 0 rz 119.57 deg; joints [25.813, -60.039, 128.834, -36.515, -72.682, 12.429]
  MoveL 553 to (237.58, 56.67, 0) mm, rotated rx -180 ry 0 rz 119.57 deg; joints [24.822, -58.23, 125.244, -37.878, -71.489, 13.873]
  MoveL 554 to (237.58, 148.11, 0) mm, rotated rx 180 ry 0 rz 119.57 deg; joints [20.907, -59.663, 128.088, -41.576, -73.522, 14.124]
  MoveL 555 to (222.3, 148.11, 0) mm, rotated rx -180 ry 0 rz 119.57 deg; joints [21.167, -60.232, 129.218, -41.205, -73.88, 13.664]
  MoveL 556 to (222.3, 75.72, 0) mm, rotated rx -180 ry 0 rz 119.57 deg; joints [24.315, -59.112, 126.995, -38.221, -72.293, 13.47]
  MoveL 557 to (222.25, 74.93, 0) mm, rotated rx 180 ry 0 rz 119.57 deg; joints [24.349, -59.1, 126.972, -38.188, -72.276, 13.467]
  MoveL 558 to (222.12, 74.16, 0) mm, rotated rx -180 ry 0 rz 119.57 deg; joints [24.384, -59.092, 126.957, -38.154, -72.262, 13.461]
  MoveL 559 to (221.91, 73.42, 0) mm, rotated rx -180 ry 0 rz 119.57 deg; joints [24.42, -59.088, 126.947, -38.118, -72.25, 13.453]
  MoveL 560 to (221.62, 72.7, 0) mm, rotated rx -180 ry 0 rz 119.57 deg; joints [24.456, -59.086, 126.945, -38.082, -72.241, 13.442]
  MoveL 561 to (221.25, 72.02, 0) mm, rotated rx -180 ry 0 rz 119.57 deg; joints [24.492, -59.088, 126.949, -38.045, -72.234, 13.43]
  MoveL 562 to (220.82, 71.38, 0) mm, rotated rx -180 ry 0 rz 119.57 deg; joints [24.528, -59.094, 126.959, -38.008, -72.23, 13.415]
  MoveL 563 to (220.32, 70.78, 0) mm, rotated rx 180 ry 0 rz 119.57 deg; joints [24.563, -59.102, 126.976, -37.97, -72.228, 13.399]
  MoveL 564 to (219.76, 70.23, 0) mm, rotated rx -180 ry 0 rz 119.57 deg; joints [24.597, -59.113, 126.998, -37.933, -72.229, 13.381]
  MoveL 565 to (219.14, 69.74, 0) mm, rotated rx -180 ry 0 rz 119.57 deg; joints [24.63, -59.128, 127.027, -37.897, -72.232, 13.362]
  MoveL 566 to (218.49, 69.31, 0) mm, rotated rx 180 ry 0 rz 119.57 deg; joints [24.661, -59.144, 127.06, -37.862, -72.238, 13.342]
  MoveL 567 to (217.79, 68.94, 0) mm, rotated rx 180 ry 0 rz 119.57 deg; joints [24.69, -59.163, 127.098, -37.828, -72.246, 13.32]
  MoveL 568 to (217.07, 68.64, 0) mm, rotated rx 180 ry 0 rz 119.57 deg; joints [24.716, -59.185, 127.14, -37.797, -72.257, 13.299]
  MoveL 569 to (216.33, 68.4, 0) mm, rotated rx 180 ry 0 rz 119.57 deg; joints [24.741, -59.208, 127.186, -37.767, -72.269, 13.276]
  MoveL 570 to (215.56, 68.23, 0) mm, rotated rx -180 ry 0 rz 119.57 deg; joints [24.763, -59.233, 127.236, -37.74, -72.284, 13.253]
  MoveL 571 to (214.78, 68.13, 0) mm, rotated rx 180 ry 0 rz 119.57 deg; joints [24.783, -59.26, 127.289, -37.715, -72.3, 13.23]
  Set speed (2000.0 mm/s)
  MoveL 572 to (214.78, 68.13, 0) mm, rotated rx 180 ry 0 rz 119.57 deg; joints [24.783, -59.26, 127.289, -37.715, -72.3, 13.23]
  MoveL 573 to (214.78, 68.13, 10) mm, rotated rx -180 ry 0 rz 119.57 deg; joints [24.783, -59.9, 127.262, -37.847, -71.772, 13.66]
  Set speed (2000.0 mm/s)
  MoveL 574 to (133.29, 103.36, 0) mm, rotated rx -180 ry 0 rz 119.57 deg; joints [24.892, -62.77, 134.242, -36.99, -75.014, 11.022]
  MoveL 575 to (133.29, 103.36, 0) mm, rotated rx -180 ry 0 rz 119.57 deg; joints [24.892, -62.77, 134.242, -36.99, -75.014, 11.022]
  Set speed (60.0 mm/s)
  MoveL 576 to (132.69, 104.21, 0) mm, rotated rx 180 ry 0 rz 119.57 deg; joints [24.866, -62.805, 134.312, -37.011, -75.047, 11.007]
  MoveL 577 to (132.03, 105.02, 0) mm, rotated rx 180 ry 0 rz 119.57 deg; joints [24.843, -62.841, 134.384, -37.029, -75.08, 10.991]
  MoveL 578 to (130.56, 106.48, 0) mm, rotated rx 180 ry 0 rz 119.57 deg; joints [24.807, -62.917, 134.534, -37.053, -75.146, 10.954]
  MoveL 579 to (128.91, 107.75, 0) mm, rotated rx -180 ry 0 rz 119.57 deg; joints [24.784, -62.996, 134.69, -37.065, -75.212, 10.912]
  MoveL 580 to (127.11, 108.8, 0) mm, rotated rx -180 ry 0 rz 119.57 deg; joints [24.774, -63.077, 134.85, -37.063, -75.277, 10.866]
  MoveL 581 to (125.21, 109.63, 0) mm, rotated rx -180 ry 0 rz 119.57 deg; joints [24.776, -63.157, 135.009, -37.048, -75.339, 10.816]
  MoveL 582 to (123.22, 110.22, 0) mm, rotated rx 180 ry 0 rz 119.57 deg; joints [24.791, -63.237, 135.166, -37.02, -75.398, 10.764]
  MoveL 583 to (121.18, 110.57, 0) mm, rotated rx 180 ry 0 rz 119.57 deg; joints [24.819, -63.315, 135.32, -36.981, -75.454, 10.71]
  MoveL 584 to (119.11, 110.69, 0) mm, rotated rx 180 ry 0 rz 119.57 deg; joints [24.857, -63.39, 135.468, -36.93, -75.505, 10.655]
  MoveL 585 to (67.1, 110.69, 0) mm, rotated rx 180 ry 0 rz 119.57 deg; joints [26.024, -65.199, 139.037, -35.489, -76.723, 9.3]
  MoveL 586 to (67.1, 122.12, 0) mm, rotated rx 180 ry 0 rz 119.57 deg; joints [25.473, -65.389, 139.412, -36.022, -76.962, 9.316]
  MoveL 587 to (135.45, 122.12, 0) mm, rotated rx 180 ry 0 rz 119.57 deg; joints [23.984, -62.995, 134.688, -37.877, -75.364, 11.119]
  MoveL 588 to (185.81, 45.92, 0) mm, rotated rx -180 ry 0 rz 119.57 deg; joints [26.314, -59.923, 128.605, -36.024, -72.483, 12.346]
  MoveL 589 to (171.25, 45.92, 0) mm, rotated rx -180 ry 0 rz 119.57 deg; joints [26.623, -60.442, 129.635, -35.614, -72.832, 11.938]
  MoveL 590 to (133.29, 103.36, 0) mm, rotated rx -180 ry 0 rz 119.57 deg; joints [24.892, -62.77, 134.242, -36.99, -75.014, 11.022]
  Set speed (2000.0 mm/s)
  MoveL 591 to (133.29, 103.36, 0) mm, rotated rx -180 ry 0 rz 119.57 deg; joints [24.892, -62.77, 134.242, -36.99, -75.014, 11.022]
  MoveL 592 to (133.29, 103.36, 10) mm, rotated rx -180 ry 0 rz 119.57 deg; joints [24.892, -63.483, 134.213, -37.112, -74.422, 11.486]
  Set speed (2000.0 mm/s)
  MoveL 593 to (237.58, 26.87, 0) mm, rotated rx -180 ry 0 rz 119.57 deg; joints [26.048, -57.709, 124.209, -36.727, -70.787, 13.795]
  MoveL 594 to (237.58, 26.87, 0) mm, rotated rx -180 ry 0 rz 119.57 deg; joints [26.048, -57.709, 124.209, -36.727, -70.787, 13.795]
  Set speed (60.0 mm/s)
  MoveL 595 to (237.58, 38.3, 0) mm, rotated rx 180 ry 0 rz 119.57 deg; joints [25.58, -57.912, 124.612, -37.165, -71.058, 13.825]
  MoveL 596 to (170.8, 38.3, 0) mm, rotated rx -180 ry 0 rz 119.57 deg; joints [26.958, -60.322, 129.396, -35.292, -72.666, 11.908]
  MoveL 597 to (166.69, 38.78, 0) mm, rotated rx 180 ry 0 rz 119.57 deg; joints [27.027, -60.476, 129.702, -35.194, -72.776, 11.796]
  MoveL 598 to (164.7, 39.37, 0) mm, rotated rx -180 ry 0 rz 119.57 deg; joints [27.045, -60.557, 129.862, -35.161, -72.837, 11.742]
  MoveL 599 to (162.79, 40.19, 0) mm, rotated rx 180 ry 0 rz 119.57 deg; joints [27.052, -60.639, 130.025, -35.14, -72.902, 11.692]
  MoveL 600 to (161, 41.25, 0) mm, rotated rx 180 ry 0 rz 119.57 deg; joints [27.046, -60.722, 130.189, -35.132, -72.969, 11.645]
  MoveL 601 to (159.35, 42.51, 0) mm, rotated rx 180 ry 0 rz 119.57 deg; joints [27.028, -60.803, 130.349, -35.137, -73.038, 11.602]
  MoveL 602 to (157.88, 43.98, 0) mm, rotated rx -180 ry 0 rz 119.57 deg; joints [26.997, -60.881, 130.504, -35.155, -73.107, 11.565]
  MoveL 603 to (156.61, 45.64, 0) mm, rotated rx -180 ry 0 rz 119.57 deg; joints [26.953, -60.955, 130.651, -35.187, -73.176, 11.534]
  MoveL 604 to (118.65, 103.07, 0) mm, rotated rx -180 ry 0 rz 119.57 deg; joints [25.22, -63.281, 135.252, -36.578, -75.353, 10.628]
  MoveL 605 to (104.09, 103.07, 0) mm, rotated rx -180 ry 0 rz 119.57 deg; joints [25.54, -63.79, 136.259, -36.177, -75.695, 10.242]
  MoveL 606 to (154.45, 26.87, 0) mm, rotated rx 180 ry 0 rz 119.57 deg; joints [27.805, -60.69, 130.125, -34.359, -72.792, 11.434]
  MoveL 607 to (237.58, 26.87, 0) mm, rotated rx -180 ry 0 rz 119.57 deg; joints [26.048, -57.709, 124.209, -36.727, -70.787, 13.795]
  Set speed (2000.0 mm/s)
  MoveL 608 to (237.58, 26.87, 0) mm, rotated rx -180 ry 0 rz 119.57 deg; joints [26.048, -57.709, 124.209, -36.727, -70.787, 13.795]
  MoveL 609 to (237.58, 26.87, 10) mm, rotated rx -180 ry 0 rz 119.57 deg; joints [26.048, -58.323, 124.183, -36.862, -70.274, 14.201]
  Set speed (2000.0 mm/s)
  MoveL 610 to (268, 87.6, 0) mm, rotated rx -180 ry 0 rz 119.57 deg; joints [22.974, -57.607, 124.007, -39.895, -71.469, 14.879]
  MoveL 611 to (268, 87.6, 0) mm, rotated rx -180 ry 0 rz 119.57 deg; joints [22.974, -57.607, 124.007, -39.895, -71.469, 14.879]
  Set speed (60.0 mm/s)
  MoveL 612 to (267.22, 87.49, 0) mm, rotated rx -180 ry 0 rz 119.57 deg; joints [22.992, -57.635, 124.062, -39.871, -71.486, 14.855]
  MoveL 613 to (266.46, 87.32, 0) mm, rotated rx -180 ry 0 rz 119.57 deg; joints [23.012, -57.661, 124.114, -39.845, -71.5, 14.831]
  MoveL 614 to (265.71, 87.09, 0) mm, rotated rx -180 ry 0 rz 119.57 deg; joints [23.035, -57.685, 124.162, -39.816, -71.513, 14.807]
  MoveL 615 to (264.99, 86.79, 0) mm, rotated rx -180 ry 0 rz 119.57 deg; joints [23.061, -57.708, 124.206, -39.785, -71.523, 14.784]
  MoveL 616 to (264.3, 86.42, 0) mm, rotated rx 180 ry 0 rz 119.57 deg; joints [23.088, -57.728, 124.246, -39.753, -71.531, 14.762]
  MoveL 617 to (263.64, 85.99, 0) mm, rotated rx 180 ry 0 rz 119.57 deg; joints [23.118, -57.745, 124.282, -39.719, -71.537, 14.74]
  MoveL 618 to (263.03, 85.5, 0) mm, rotated rx 180 ry 0 rz 119.57 deg; joints [23.15, -57.761, 124.312, -39.684, -71.541, 14.72]
  MoveL 619 to (262.46, 84.95, 0) mm, rotated rx -180 ry 0 rz 119.57 deg; joints [23.183, -57.773, 124.336, -39.647, -71.542, 14.701]
  MoveL 620 to (261.96, 84.35, 0) mm, rotated rx -180 ry 0 rz 119.57 deg; joints [23.217, -57.782, 124.354, -39.611, -71.54, 14.684]
  MoveL 621 to (261.53, 83.71, 0) mm, rotated rx 180 ry 0 rz 119.57 deg; joints [23.251, -57.788, 124.366, -39.574, -71.536, 14.669]
  MoveL 622 to (261.17, 83.02, 0) mm, rotated rx 180 ry 0 rz 119.57 deg; joints [23.286, -57.791, 124.371, -39.538, -71.529, 14.656]
  MoveL 623 to (260.88, 82.31, 0) mm, rotated rx -180 ry 0 rz 119.57 deg; joints [23.321, -57.79, 124.37, -39.503, -71.52, 14.645]
  MoveL 624 to (260.66, 81.57, 0) mm, rotated rx 180 ry 0 rz 119.57 deg; joints [23.356, -57.786, 124.362, -39.468, -71.508, 14.637]
  MoveL 625 to (260.53, 80.8, 0) mm, rotated rx -180 ry 0 rz 119.57 deg; joints [23.39, -57.778, 124.347, -39.435, -71.493, 14.631]
  MoveL 626 to (260.49, 80.01, 0) mm, rotated rx 180 ry 0 rz 119.57 deg; joints [23.424, -57.767, 124.325, -39.403, -71.476, 14.627]
  MoveL 627 to (260.49, 7.62, 0) mm, rotated rx 180 ry 0 rz 119.57 deg; joints [26.368, -56.516, 121.836, -36.649, -69.763, 14.432]
  MoveL 628 to (245.2, 7.62, 0) mm, rotated rx -180 ry 0 rz 119.57 deg; joints [26.672, -57.079, 122.957, -36.214, -70.137, 13.972]
  MoveL 629 to (245.2, 99.06, 0) mm, rotated rx 180 ry 0 rz 119.57 deg; joints [22.897, -58.642, 126.063, -39.759, -72.273, 14.215]
  MoveL 630 to (294.94, 99.06, 0) mm, rotated rx -180 ry 0 rz 119.57 deg; joints [22.036, -56.766, 122.335, -41.033, -71.085, 15.755]
  MoveL 631 to (335.23, 38.1, 0) mm, rotated rx -180 ry 0 rz 119.57 deg; joints [23.796, -54.221, 117.269, -39.833, -68.671, 16.878]
  MoveL 632 to (320.67, 38.1, 0) mm, rotated rx -180 ry 0 rz 119.57 deg; joints [24.048, -54.784, 118.391, -39.436, -69.029, 16.402]
  MoveL 633 to (290.35, 83.96, 0) mm, rotated rx -180 ry 0 rz 119.57 deg; joints [22.735, -56.704, 122.211, -40.336, -70.849, 15.566]
  MoveL 634 to (289.72, 84.8, 0) mm, rotated rx -180 ry 0 rz 119.57 deg; joints [22.711, -56.741, 122.286, -40.351, -70.884, 15.548]
  MoveL 635 to (288.98, 85.53, 0) mm, rotated rx -180 ry 0 rz 119.57 deg; joints [22.694, -56.781, 122.365, -40.36, -70.919, 15.527]
  MoveL 636 to (288.16, 86.16, 0) mm, rotated rx -180 ry 0 rz 119.57 deg; joints [22.682, -56.822, 122.447, -40.363, -70.953, 15.503]
  MoveL 637 to (287.27, 86.68, 0) mm, rotated rx -180 ry 0 rz 119.57 deg; joints [22.676, -56.864, 122.53, -40.36, -70.986, 15.476]
  MoveL 638 to (286.32, 87.09, 0) mm, rotated rx -180 ry 0 rz 119.57 deg; joints [22.675, -56.907, 122.615, -40.351, -71.018, 15.448]
  MoveL 639 to (285.32, 87.39, 0) mm, rotated rx 180 ry 0 rz 119.57 deg; joints [22.68, -56.949, 122.699, -40.337, -71.049, 15.417]
  MoveL 640 to (284.3, 87.57, 0) mm, rotated rx 180 ry 0 rz 119.57 deg; joints [22.69, -56.991, 122.782, -40.317, -71.078, 15.386]
  MoveL 641 to (283.26, 87.63, 0) mm, rotated rx -180 ry 0 rz 119.57 deg; joints [22.706, -57.032, 122.863, -40.292, -71.104, 15.353]
  MoveL 642 to (268.79, 87.63, 0) mm, rotated rx -180 ry 0 rz 119.57 deg; joints [22.959, -57.578, 123.95, -39.917, -71.451, 14.903]
  MoveL 643 to (268, 87.6, 0) mm, rotated rx -180 ry 0 rz 119.57 deg; joints [22.974, -57.607, 124.007, -39.895, -71.469, 14.879]
  Set speed (2000.0 mm/s)
  MoveL 644 to (268, 87.6, 0) mm, rotated rx -180 ry 0 rz 119.57 deg; joints [22.974, -57.607, 124.007, -39.895, -71.469, 14.879]
  MoveL 645 to (268, 87.6, 10) mm, rotated rx -180 ry 0 rz 119.57 deg; joints [22.974, -58.219, 123.981, -40.035, -70.98, 15.312]
  Set speed (2000.0 mm/s)
  MoveL 646 to (335.34, 19.08, 0) mm, rotated rx -180 ry 0 rz 119.57 deg; joints [24.529, -53.885, 116.6, -39.162, -68.202, 16.828]
  MoveL 647 to (335.34, 19.08, 0) mm, rotated rx -180 ry 0 rz 119.57 deg; joints [24.529, -53.885, 116.6, -39.162, -68.202, 16.828]
  Set speed (60.0 mm/s)
  MoveL 648 to (334.56, 19.05, 0) mm, rotated rx 180 ry 0 rz 119.57 deg; joints [24.544, -53.915, 116.66, -39.139, -68.22, 16.802]
  MoveL 649 to (320.08, 19.05, 0) mm, rotated rx 180 ry 0 rz 119.57 deg; joints [24.801, -54.474, 117.773, -38.737, -68.578, 16.33]
  MoveL 650 to (318.02, 19.29, 0) mm, rotated rx -180 ry 0 rz 119.57 deg; joints [24.828, -54.557, 117.939, -38.688, -68.635, 16.264]
  MoveL 651 to (317.03, 19.59, 0) mm, rotated rx 180 ry 0 rz 119.57 deg; joints [24.835, -54.601, 118.025, -38.671, -68.667, 16.233]
  MoveL 652 to (316.08, 20, 0) mm, rotated rx -180 ry 0 rz 119.57 deg; joints [24.836, -54.644, 118.112, -38.659, -68.7, 16.203]
  MoveL 653 to (315.18, 20.52, 0) mm, rotated rx 180 ry 0 rz 119.57 deg; joints [24.832, -54.688, 118.199, -38.653, -68.735, 16.176]
  MoveL 654 to (314.36, 21.15, 0) mm, rotated rx -180 ry 0 rz 119.57 deg; joints [24.822, -54.73, 118.284, -38.653, -68.771, 16.151]
  MoveL 655 to (313.63, 21.88, 0) mm, rotated rx 180 ry 0 rz 119.57 deg; joints [24.807, -54.772, 118.366, -38.659, -68.807, 16.13]
  MoveL 656 to (312.99, 22.72, 0) mm, rotated rx -180 ry 0 rz 119.57 deg; joints [24.786, -54.811, 118.444, -38.671, -68.843, 16.112]
  MoveL 657 to (282.68, 68.58, 0) mm, rotated rx 180 ry 0 rz 119.57 deg; joints [23.498, -56.746, 122.295, -39.547, -70.678, 15.28]
  MoveL 658 to (268.12, 68.58, 0) mm, rotated rx -180 ry 0 rz 119.57 deg; joints [23.759, -57.294, 123.385, -39.161, -71.03, 14.829]
  MoveL 659 to (308.41, 7.62, 0) mm, rotated rx -180 ry 0 rz 119.57 deg; joints [25.456, -54.716, 118.254, -38.003, -68.584, 15.924]
  MoveL 660 to (358.14, 7.62, 0) mm, rotated rx -180 ry 0 rz 119.57 deg; joints [24.569, -52.791, 114.419, -39.402, -67.348, 17.556]
  MoveL 661 to (358.14, 99.06, 0) mm, rotated rx -180 ry 0 rz 119.57 deg; joints [21.026, -54.308, 117.443, -42.641, -69.563, 17.825]
  MoveL 662 to (342.85, 99.06, 0) mm, rotated rx -180 ry 0 rz 119.57 deg; joints [21.262, -54.911, 118.643, -42.252, -69.932, 17.312]
  MoveL 663 to (342.85, 26.67, 0) mm, rotated rx -180 ry 0 rz 119.57 deg; joints [24.107, -53.727, 116.284, -39.637, -68.203, 17.097]
  MoveL 664 to (342.81, 25.88, 0) mm, rotated rx 180 ry 0 rz 119.57 deg; joints [24.138, -53.715, 116.26, -39.609, -68.185, 17.094]
  MoveL 665 to (342.68, 25.11, 0) mm, rotated rx -180 ry 0 rz 119.57 deg; joints [24.169, -53.706, 116.243, -39.578, -68.169, 17.087]
  MoveL 666 to (342.47, 24.37, 0) mm, rotated rx -180 ry 0 rz 119.57 deg; joints [24.202, -53.702, 116.234, -39.546, -68.156, 17.078]
  MoveL 667 to (342.18, 23.65, 0) mm, rotated rx 180 ry 0 rz 119.57 deg; joints [24.234, -53.7, 116.231, -39.513, -68.145, 17.066]
  MoveL 668 to (341.81, 22.97, 0) mm, rotated rx 180 ry 0 rz 119.57 deg; joints [24.267, -53.703, 116.236, -39.479, -68.138, 17.053]
  MoveL 669 to (341.38, 22.33, 0) mm, rotated rx -180 ry 0 rz 119.57 deg; joints [24.299, -53.708, 116.247, -39.444, -68.133, 17.036]
  MoveL 670 to (340.88, 21.73, 0) mm, rotated rx 180 ry 0 rz 119.57 deg; joints [24.331, -53.717, 116.265, -39.409, -68.13, 17.018]
  MoveL 671 to (340.32, 21.18, 0) mm, rotated rx -180 ry 0 rz 119.57 deg; joints [24.361, -53.729, 116.289, -39.374, -68.13, 16.998]
  MoveL 672 to (339.7, 20.69, 0) mm, rotated rx 180 ry 0 rz 119.57 deg; joints [24.391, -53.745, 116.32, -39.34, -68.134, 16.976]
  MoveL 673 to (339.04, 20.26, 0) mm, rotated rx 180 ry 0 rz 119.57 deg; joints [24.419, -53.763, 116.355, -39.307, -68.139, 16.953]
  MoveL 674 to (338.35, 19.89, 0) mm, rotated rx 180 ry 0 rz 119.57 deg; joints [24.445, -53.783, 116.396, -39.275, -68.147, 16.93]
  MoveL 675 to (337.63, 19.59, 0) mm, rotated rx 180 ry 0 rz 119.57 deg; joints [24.469, -53.806, 116.441, -39.244, -68.158, 16.905]
  MoveL 676 to (336.88, 19.36, 0) mm, rotated rx -180 ry 0 rz 119.57 deg; joints [24.491, -53.83, 116.491, -39.215, -68.17, 16.88]
  MoveL 677 to (336.12, 19.19, 0) mm, rotated rx 180 ry 0 rz 119.57 deg; joints [24.511, -53.857, 116.544, -39.188, -68.185, 16.854]
  MoveL 678 to (335.34, 19.08, 0) mm, rotated rx -180 ry 0 rz 119.57 deg; joints [24.529, -53.885, 116.6, -39.162, -68.202, 16.828]
  Set speed (2000.0 mm/s)
  MoveL 679 to (335.34, 19.08, 0) mm, rotated rx -180 ry 0 rz 119.57 deg; joints [24.529, -53.885, 116.6, -39.162, -68.202, 16.828]
  MoveL 680 to (335.34, 19.08, 10) mm, rotated rx -180 ry 0 rz 119.57 deg; joints [24.529, -54.443, 116.576, -39.311, -67.751, 17.225]
  Set speed (2000.0 mm/s)
  MoveL 681 to (232.4, 7.62, 0) mm, rotated rx 180 ry 0 rz 119.57 deg; joints [26.932, -57.548, 123.888, -35.849, -70.449, 13.593]
  MoveL 682 to (232.4, 7.62, 0) mm, rotated rx 180 ry 0 rz 119.57 deg; joints [26.932, -57.548, 123.888, -35.849, -70.449, 13.593]
  Set speed (60.0 mm/s)
  MoveL 683 to (139.42, 7.62, 0) mm, rotated rx -180 ry 0 rz 119.57 deg; joints [28.967, -60.851, 130.445, -33.138, -72.697, 10.988]
  MoveL 684 to (89.06, 83.82, 0) mm, rotated rx -180 ry 0 rz 119.57 deg; joints [26.776, -63.984, 136.641, -34.893, -75.633, 9.818]
  MoveL 685 to (103.62, 83.82, 0) mm, rotated rx 180 ry 0 rz 119.57 deg; joints [26.44, -63.48, 135.646, -35.308, -75.29, 10.195]
  MoveL 686 to (141.58, 26.38, 0) mm, rotated rx -180 ry 0 rz 119.57 deg; joints [28.119, -61.131, 130.998, -33.963, -73.088, 11.086]
  MoveL 687 to (142.84, 24.73, 0) mm, rotated rx -180 ry 0 rz 119.57 deg; joints [28.16, -61.056, 130.85, -33.932, -73.019, 11.116]
  MoveL 688 to (144.31, 23.26, 0) mm, rotated rx 180 ry 0 rz 119.57 deg; joints [28.19, -60.977, 130.694, -33.916, -72.95, 11.153]
  MoveL 689 to (145.96, 21.99, 0) mm, rotated rx -180 ry 0 rz 119.57 deg; joints [28.206, -60.896, 130.534, -33.913, -72.881, 11.194]
  MoveL 690 to (147.76, 20.94, 0) mm, rotated rx -180 ry 0 rz 119.57 deg; joints [28.21, -60.813, 130.37, -33.923, -72.813, 11.24]
  MoveL 691 to (149.66, 20.12, 0) mm, rotated rx 180 ry 0 rz 119.57 deg; joints [28.201, -60.731, 130.208, -33.945, -72.748, 11.29]
  MoveL 692 to (151.65, 19.53, 0) mm, rotated rx 180 ry 0 rz 119.57 deg; joints [28.181, -60.651, 130.048, -33.98, -72.686, 11.342]
  MoveL 693 to (155.76, 19.05, 0) mm, rotated rx -180 ry 0 rz 119.57 deg; joints [28.108, -60.498, 129.745, -34.081, -72.576, 11.453]
  MoveL 694 to (232.4, 19.05, 0) mm, rotated rx 180 ry 0 rz 119.57 deg; joints [26.47, -57.757, 124.305, -36.282, -70.725, 13.622]
  MoveL 695 to (232.4, 7.62, 0) mm, rotated rx 180 ry 0 rz 119.57 deg; joints [26.932, -57.548, 123.888, -35.849, -70.449, 13.593]
  Set speed (2000.0 mm/s)
  MoveL 696 to (232.4, 7.62, 0) mm, rotated rx 180 ry 0 rz 119.57 deg; joints [26.932, -57.548, 123.888, -35.849, -70.449, 13.593]
  MoveL 697 to (232.4, 7.62, 10) mm, rotated rx -180 ry 0 rz 119.57 deg; joints [26.932, -58.159, 123.862, -35.984, -69.933, 13.99]
  Set speed (2000.0 mm/s)
  MoveL 698 to (298.33, 121.92, 0) mm, rotated rx -180 ry 0 rz 119.57 deg; joints [21.032, -56.982, 122.763, -42.005, -71.518, 15.933]
  MoveL 699 to (298.33, 121.92, 0) mm, rotated rx -180 ry 0 rz 119.57 deg; joints [21.032, -56.982, 122.763, -42.005, -71.518, 15.933]
  Set speed (60.0 mm/s)
  MoveL 700 to (308.41, 106.68, 0) mm, rotated rx -180 ry 0 rz 119.57 deg; joints [21.5, -56.366, 121.539, -41.668, -70.935, 16.209]
  MoveL 701 to (320.84, 106.68, 0) mm, rotated rx -180 ry 0 rz 119.57 deg; joints [21.301, -55.885, 120.583, -41.981, -70.637, 16.611]
  MoveL 702 to (333.27, 106.68, 0) mm, rotated rx 180 ry 0 rz 119.57 deg; joints [21.105, -55.402, 119.62, -42.294, -70.338, 17.019]
  MoveL 703 to (345.71, 106.68, 0) mm, rotated rx 180 ry 0 rz 119.57 deg; joints [20.912, -54.914, 118.65, -42.607, -70.039, 17.432]
  MoveL 704 to (358.14, 106.68, 0) mm, rotated rx -180 ry 0 rz 119.57 deg; joints [20.723, -54.424, 117.672, -42.92, -69.739, 17.85]
  MoveL 705 to (358.14, 129.54, 0) mm, rotated rx -180 ry 0 rz 119.57 deg; joints [19.805, -54.758, 118.339, -43.766, -70.262, 17.925]
  MoveL 706 to (358.14, 152.4, 0) mm, rotated rx 180 ry 0 rz 119.57 deg; joints [18.877, -55.077, 118.973, -44.625, -70.775, 18.004]
  MoveL 707 to (358.14, 175.26, 0) mm, rotated rx -180 ry 0 rz 119.57 deg; joints [17.938, -55.38, 119.576, -45.496, -71.278, 18.086]
  MoveL 708 to (358.14, 198.12, 0) mm, rotated rx 180 ry 0 rz 119.57 deg; joints [16.99, -55.667, 120.147, -46.378, -71.771, 18.172]
  MoveL 709 to (342.85, 198.12, 0) mm, rotated rx -180 ry 0 rz 119.57 deg; joints [17.187, -56.274, 121.356, -46.04, -72.126, 17.654]
  MoveL 710 to (342.85, 125.73, 0) mm, rotated rx -180 ry 0 rz 119.57 deg; joints [20.185, -55.307, 119.432, -43.249, -70.542, 17.398]
  MoveL 711 to (342.81, 124.94, 0) mm, rotated rx 180 ry 0 rz 119.57 deg; joints [20.218, -55.298, 119.413, -43.218, -70.525, 17.394]
  MoveL 712 to (342.68, 124.17, 0) mm, rotated rx -180 ry 0 rz 119.57 deg; joints [20.251, -55.292, 119.401, -43.186, -70.511, 17.387]
  MoveL 713 to (342.47, 123.43, 0) mm, rotated rx -180 ry 0 rz 119.57 deg; joints [20.284, -55.289, 119.396, -43.153, -70.499, 17.378]
  MoveL 714 to (342.18, 122.71, 0) mm, rotated rx -180 ry 0 rz 119.57 deg; joints [20.318, -55.29, 119.398, -43.119, -70.49, 17.366]
  MoveL 715 to (341.81, 122.03, 0) mm, rotated rx 180 ry 0 rz 119.57 deg; joints [20.351, -55.295, 119.407, -43.084, -70.483, 17.352]
  MoveL 716 to (341.38, 121.39, 0) mm, rotated rx -180 ry 0 rz 119.57 deg; joints [20.384, -55.302, 119.422, -43.049, -70.479, 17.335]
  MoveL 717 to (340.88, 120.79, 0) mm, rotated rx 180 ry 0 rz 119.57 deg; joints [20.415, -55.313, 119.444, -43.014, -70.478, 17.316]
  MoveL 718 to (340.32, 120.24, 0) mm, rotated rx 180 ry 0 rz 119.57 deg; joints [20.446, -55.327, 119.472, -42.98, -70.479, 17.296]
  MoveL 719 to (339.7, 119.75, 0) mm, rotated rx -180 ry 0 rz 119.57 deg; joints [20.476, -55.344, 119.506, -42.946, -70.482, 17.274]
